    p_a_dep_fam_3:
        !Ponto antes de depositar
        pMov_Pega_Depos_Buffer := pPosição_Final_Buffer;
        pMov_Pega_Depos_Buffer.trans := pMov_Pega_Depos_Buffer.trans + pOfst_Z_Familia_3;
        IF (nPos_Buffer >= 13 AND nPos_Buffer <= 15) OR (nPos_Buffer >= 19 AND nPos_Buffer <= 21) OR (nPos_Buffer >= 25 AND nPos_Buffer <= 27) OR (nPos_Buffer >= 31 AND nPos_Buffer <=33) OR (nPos_Buffer >= 37 AND nPos_Buffer <= 39) OR (nPos_Buffer >= 43 AND nPos_Buffer <= 45) OR (nPos_Buffer >= 49 AND nPos_Buffer <= 51) OR (nPos_Buffer >= 55 AND nPos_Buffer <=57) OR (nPos_Buffer >= 61 AND nPos_Buffer <= 63) OR (nPos_Buffer >= 67 AND nPos_Buffer <= 69) OR (nPos_Buffer >= 73 AND nPos_Buffer <= 75) OR (nPos_Buffer >= 79 AND nPos_Buffer <= 81) OR (nPos_Buffer >= 85 AND nPos_Buffer <= 87) OR (nPos_Buffer >= 91 AND nPos_Buffer <= 93) OR (nPos_Buffer >= 97 AND nPos_Buffer <= 99) THEN
        MoveL pMov_Pega_Depos_Buffer, SMov_SuperFina, z10, tGarra \WObj:=wBuffer_Dir;
        GOTO p_ant_ag_3;
        ENDIF
        IF (nPos_Buffer >= 1 AND nPos_Buffer <= 9) THEN
        MoveL pMov_Pega_Depos_Buffer, SMov_SuperFina, z10, tGarra \WObj:=wBuffer_Front;
        GOTO p_ant_ag_3;
        ELSE
        MoveL pMov_Pega_Depos_Buffer, SMov_SuperFina, z10, tGarra \WObj:=wBuffer_Esq;
        ENDIF

    p_ant_ag_3:
        pMov_Pega_Depos_Buffer := pPosição_Final_Buffer;
        pMov_Pega_Depos_Buffer.trans := pMov_Pega_Depos_Buffer.trans + pOfst_Aprox_Final_Depos;
        IF (nPos_Buffer >= 13 AND nPos_Buffer <= 15) OR (nPos_Buffer >= 19 AND nPos_Buffer <= 21) OR (nPos_Buffer >= 25 AND nPos_Buffer <= 27) OR (nPos_Buffer >= 31 AND nPos_Buffer <=33) OR (nPos_Buffer >= 37 AND nPos_Buffer <= 39) OR (nPos_Buffer >= 43 AND nPos_Buffer <= 45) OR (nPos_Buffer >= 49 AND nPos_Buffer <= 51) OR (nPos_Buffer >= 55 AND nPos_Buffer <=57) OR (nPos_Buffer >= 61 AND nPos_Buffer <= 63) OR (nPos_Buffer >= 67 AND nPos_Buffer <= 69) OR (nPos_Buffer >= 73 AND nPos_Buffer <= 75) OR (nPos_Buffer >= 79 AND nPos_Buffer <= 81) OR (nPos_Buffer >= 85 AND nPos_Buffer <= 87) OR (nPos_Buffer >= 91 AND nPos_Buffer <= 93) OR (nPos_Buffer >= 97 AND nPos_Buffer <= 99) THEN
        MoveL pMov_Pega_Depos_Buffer, SMov_SuperFina, z1, tGarra \WObj:=wBuffer_Dir;
        GOTO p_depos_3;
        ENDIF
        IF (nPos_Buffer >= 1 AND nPos_Buffer <= 9) THEN
        MoveL pMov_Pega_Depos_Buffer, SMov_SuperFina, z1, tGarra \WObj:=wBuffer_Front;
        GOTO p_depos_3;
        ELSE
        MoveL pMov_Pega_Depos_Buffer, SMov_SuperFina, z1, tGarra \WObj:=wBuffer_Esq;
        ENDIF

    p_depos_3:
        !Destrava o produto
        GARRA_DestravarProduto;

        !Ponto final para depositar
        pMov_Pega_Depos_Buffer := pPosição_Final_Buffer;
        IF (nPos_Buffer >= 13 AND nPos_Buffer <= 15) OR (nPos_Buffer >= 19 AND nPos_Buffer <= 21) OR (nPos_Buffer >= 25 AND nPos_Buffer <= 27) OR (nPos_Buffer >= 31 AND nPos_Buffer <=33) OR (nPos_Buffer >= 37 AND nPos_Buffer <= 39) OR (nPos_Buffer >= 43 AND nPos_Buffer <= 45) OR (nPos_Buffer >= 49 AND nPos_Buffer <= 51) OR (nPos_Buffer >= 55 AND nPos_Buffer <=57) OR (nPos_Buffer >= 61 AND nPos_Buffer <= 63) OR (nPos_Buffer >= 67 AND nPos_Buffer <= 69) OR (nPos_Buffer >= 73 AND nPos_Buffer <= 75) OR (nPos_Buffer >= 79 AND nPos_Buffer <= 81) OR (nPos_Buffer >= 85 AND nPos_Buffer <= 87) OR (nPos_Buffer >= 91 AND nPos_Buffer <= 93) OR (nPos_Buffer >= 97 AND nPos_Buffer <= 99) THEN
        MoveL pMov_Pega_Depos_Buffer, SMov_SuperFina, fine, tGarra \WObj:=wBuffer_Dir;
        GOTO a_garra_3;
        ENDIF
        IF (nPos_Buffer >= 1 AND nPos_Buffer <= 9) THEN
        MoveL pMov_Pega_Depos_Buffer, SMov_SuperFina, fine, tGarra \WObj:=wBuffer_Front;
        GOTO a_garra_3;
        ELSE
        MoveL pMov_Pega_Depos_Buffer, SMov_SuperFina, fine, tGarra \WObj:=wBuffer_Esq;
        ENDIF


      a_garra_3:
        !Deposita Produto
        GARRA_AbrirGarra;

        GripLoad load0;

        !Movimento de Recuo
        AccSet nAcc_Mov_Geral, nRamp_Mov_Geral;
        pMov_Pega_Depos_Buffer := pPosição_Final_Buffer;
        pMov_Pega_Depos_Buffer.trans := pMov_Pega_Depos_Buffer.trans + pOfst_Acima_Berço_Buffer;
        IF (nPos_Buffer >= 13 AND nPos_Buffer <= 15) OR (nPos_Buffer >= 19 AND nPos_Buffer <= 21) OR (nPos_Buffer >= 25 AND nPos_Buffer <= 27) OR (nPos_Buffer >= 31 AND nPos_Buffer <=33) OR (nPos_Buffer >= 37 AND nPos_Buffer <= 39) OR (nPos_Buffer >= 43 AND nPos_Buffer <= 45) OR (nPos_Buffer >= 49 AND nPos_Buffer <= 51) OR (nPos_Buffer >= 55 AND nPos_Buffer <=57) OR (nPos_Buffer >= 61 AND nPos_Buffer <= 63) OR (nPos_Buffer >= 67 AND nPos_Buffer <= 69) OR (nPos_Buffer >= 73 AND nPos_Buffer <= 75) OR (nPos_Buffer >= 79 AND nPos_Buffer <= 81) OR (nPos_Buffer >= 85 AND nPos_Buffer <= 87) OR (nPos_Buffer >= 91 AND nPos_Buffer <= 93) OR (nPos_Buffer >= 97 AND nPos_Buffer <= 99) THEN
        MoveL pMov_Pega_Depos_Buffer, sMov_Aprox_Berço_Sem_Produto, z50, tGarra \WObj:=wBuffer_Dir;
        GOTO ad_buffer_3;
        ENDIF
        IF (nPos_Buffer >= 1 AND nPos_Buffer <= 9) THEN
        MoveL pMov_Pega_Depos_Buffer, sMov_Aprox_Berço_Sem_Produto, z50, tGarra \WObj:=wBuffer_Front;
        GOTO ad_buffer_3;
        ELSE
        MoveL pMov_Pega_Depos_Buffer, sMov_Aprox_Berço_Sem_Produto, z50, tGarra \WObj:=wBuffer_Esq;
        ENDIF

    ad_buffer_3:
        motionsup \On \TuneValue:= nSens_Colid_Mov_Geral;
        pMov_Pega_Depos_Buffer := pPosição_Final_Buffer;
        pMov_Pega_Depos_Buffer.trans := pMov_Pega_Depos_Buffer.trans + pOfst_Acima_Buffer_Sem_Produto;
        IF (nPos_Buffer >= 13 AND nPos_Buffer <= 15) OR (nPos_Buffer >= 19 AND nPos_Buffer <= 21) OR (nPos_Buffer >= 25 AND nPos_Buffer <= 27) OR (nPos_Buffer >= 31 AND nPos_Buffer <=33) OR (nPos_Buffer >= 37 AND nPos_Buffer <= 39) OR (nPos_Buffer >= 43 AND nPos_Buffer <= 45) OR (nPos_Buffer >= 49 AND nPos_Buffer <= 51) OR (nPos_Buffer >= 55 AND nPos_Buffer <=57) OR (nPos_Buffer >= 61 AND nPos_Buffer <= 63) OR (nPos_Buffer >= 67 AND nPos_Buffer <= 69) OR (nPos_Buffer >= 73 AND nPos_Buffer <= 75) OR (nPos_Buffer >= 79 AND nPos_Buffer <= 81) OR (nPos_Buffer >= 85 AND nPos_Buffer <= 87) OR (nPos_Buffer >= 91 AND nPos_Buffer <= 93) OR (nPos_Buffer >= 97 AND nPos_Buffer <= 99) THEN
        MoveL pMov_Pega_Depos_Buffer, sMov_Geral_Sem_Produto, z100, tGarra \WObj:=wBuffer_Dir;
        GOTO inposf_fam_3;
        ENDIF
        IF (nPos_Buffer >= 1 AND nPos_Buffer <= 9) THEN
        MoveL pMov_Pega_Depos_Buffer, sMov_Geral_Sem_Produto, z100, tGarra \WObj:=wBuffer_Front;
        GOTO inposf_fam_3;
        ELSE
        MoveL pMov_Pega_Depos_Buffer, sMov_Geral_Sem_Produto, z100, tGarra \WObj:=wBuffer_Esq;
        ENDIF
        GOTO inposf_fam_3;

inposf_fam_3:
        IF (nPos_Buffer >= 13 AND nPos_Buffer <= 15) OR (nPos_Buffer >= 19 AND nPos_Buffer <= 21) OR (nPos_Buffer >= 25 AND nPos_Buffer <= 27) OR (nPos_Buffer >= 31 AND nPos_Buffer <=33) OR (nPos_Buffer >= 37 AND nPos_Buffer <= 39) OR (nPos_Buffer >= 43 AND nPos_Buffer <= 45) OR (nPos_Buffer >= 49 AND nPos_Buffer <= 51) OR (nPos_Buffer >= 55 AND nPos_Buffer <=57) OR (nPos_Buffer >= 61 AND nPos_Buffer <= 63) OR (nPos_Buffer >= 67 AND nPos_Buffer <= 69) OR (nPos_Buffer >= 73 AND nPos_Buffer <= 75) OR (nPos_Buffer >= 79 AND nPos_Buffer <= 81) OR (nPos_Buffer >= 85 AND nPos_Buffer <= 87) OR (nPos_Buffer >= 91 AND nPos_Buffer <= 93) OR (nPos_Buffer >= 97 AND nPos_Buffer <= 99) THEN
        MoveAbsJ jposIntermedCentroMassa, sMov_Geral_Sem_Produto, z200, tGarra\WObj:=wBuffer_Dir;
        GOTO final;
        ENDIF
        IF (nPos_Buffer >= 1 AND nPos_Buffer <= 9) THEN
        MoveAbsJ jposIntermedCentroMassa, sMov_Geral_Sem_Produto, z200, tGarra\WObj:=wBuffer_Front;
        GOTO final;
        ELSE
        MoveAbsJ jposIntermedCentroMassa, sMov_Geral_Sem_Produto, z200, tGarra\WObj:=wBuffer_Esq;
        ENDIF
        GOTO final;

!*********************************************************************************************************************************************
!  PEGA PRODUTO NO BUFFER FAMILIA 3
!*********************************************************************************************************************************************

     pega_fam_3:
        !Ciclo para pegar peça no buffer

        GARRA_VerificarGarraVazia;
        !Abre Garra
        GARRA_DestravarProduto;
        GARRA_AbrirGarra;

        !Vai para posição intermediária no centro de massa
        AccSet nAcc_Mov_Geral, nRamp_Mov_Geral;

        IF (nPos_Buffer >= 13 AND nPos_Buffer <= 15) OR (nPos_Buffer >= 19 AND nPos_Buffer <= 21) OR (nPos_Buffer >= 25 AND nPos_Buffer <= 27) OR (nPos_Buffer >= 31 AND nPos_Buffer <=33) OR (nPos_Buffer >= 37 AND nPos_Buffer <= 39) OR (nPos_Buffer >= 43 AND nPos_Buffer <= 45) OR (nPos_Buffer >= 49 AND nPos_Buffer <= 51) OR (nPos_Buffer >= 55 AND nPos_Buffer <=57) OR (nPos_Buffer >= 61 AND nPos_Buffer <= 63) OR (nPos_Buffer >= 67 AND nPos_Buffer <= 69) OR (nPos_Buffer >= 73 AND nPos_Buffer <= 75) OR (nPos_Buffer >= 79 AND nPos_Buffer <= 81) OR (nPos_Buffer >= 85 AND nPos_Buffer <= 87) OR (nPos_Buffer >= 91 AND nPos_Buffer <= 93) OR (nPos_Buffer >= 97 AND nPos_Buffer <= 99) THEN
        pIntermedCentroMassa := pPosição_Final_Buffer;
	    jposIntermedCentroMassa := CalcJointT(pIntermedCentroMassa, tGarra \WObj:=wBuffer_Dir);
        jposIntermedCentroMassa.robax.rax_2 := jposRecolhidoEsteira.robax.rax_2;
        jposIntermedCentroMassa.robax.rax_3 := jposRecolhidoEsteira.robax.rax_3;
        jposIntermedCentroMassa.robax.rax_4 := jposRecolhidoEsteira.robax.rax_4;
        jposIntermedCentroMassa.robax.rax_5 := jposRecolhidoEsteira.robax.rax_5;

        MoveAbsJ jposIntermedCentroMassa, sMov_Geral_Sem_Produto, z200, tGarra\WObj:=wBuffer_Dir;
        GOTO inpegapos_fam_3;
        ENDIF

        IF (nPos_Buffer >= 1 AND nPos_Buffer <= 9) THEN
        pIntermedCentroMassa := pPosição_Final_Buffer;
	    jposIntermedCentroMassa := CalcJointT(pIntermedCentroMassa, tGarra \WObj:=wBuffer_Front);
        jposIntermedCentroMassa.robax.rax_2 := jposRecolhidoEsteira.robax.rax_2;
        jposIntermedCentroMassa.robax.rax_3 := jposRecolhidoEsteira.robax.rax_3;
        jposIntermedCentroMassa.robax.rax_4 := jposRecolhidoEsteira.robax.rax_4;
        jposIntermedCentroMassa.robax.rax_5 := jposRecolhidoEsteira.robax.rax_5;

        MoveAbsJ jposIntermedCentroMassa, sMov_Geral_Sem_Produto, z200, tGarra\WObj:=wBuffer_Front;
        GOTO inpegapos_fam_3;
        ELSE
        pIntermedCentroMassa := pPosição_Final_Buffer;
	    jposIntermedCentroMassa := CalcJointT(pIntermedCentroMassa, tGarra \WObj:=wBuffer_Esq);
        jposIntermedCentroMassa.robax.rax_2 := jposRecolhidoEsteira.robax.rax_2;
        jposIntermedCentroMassa.robax.rax_3 := jposRecolhidoEsteira.robax.rax_3;
        jposIntermedCentroMassa.robax.rax_4 := jposRecolhidoEsteira.robax.rax_4;
        jposIntermedCentroMassa.robax.rax_5 := jposRecolhidoEsteira.robax.rax_5;

        MoveAbsJ jposIntermedCentroMassa, sMov_Geral_Sem_Produto, z200, tGarra\WObj:=wBuffer_Esq;
        ENDIF

inpegapos_fam_3:
        !Ponto acima da posição
        pMov_Pega_Depos_Buffer := pPosição_Final_Buffer;
        pMov_Pega_Depos_Buffer.trans := pMov_Pega_Depos_Buffer.trans + pOfst_Acima_Buffer_Sem_Produto;
        IF (nPos_Buffer >= 13 AND nPos_Buffer <= 15) OR (nPos_Buffer >= 19 AND nPos_Buffer <= 21) OR (nPos_Buffer >= 25 AND nPos_Buffer <= 27) OR (nPos_Buffer >= 31 AND nPos_Buffer <=33) OR (nPos_Buffer >= 37 AND nPos_Buffer <= 39) OR (nPos_Buffer >= 43 AND nPos_Buffer <= 45) OR (nPos_Buffer >= 49 AND nPos_Buffer <= 51) OR (nPos_Buffer >= 55 AND nPos_Buffer <=57) OR (nPos_Buffer >= 61 AND nPos_Buffer <= 63) OR (nPos_Buffer >= 67 AND nPos_Buffer <= 69) OR (nPos_Buffer >= 73 AND nPos_Buffer <= 75) OR (nPos_Buffer >= 79 AND nPos_Buffer <= 81) OR (nPos_Buffer >= 85 AND nPos_Buffer <= 87) OR (nPos_Buffer >= 91 AND nPos_Buffer <= 93) OR (nPos_Buffer >= 97 AND nPos_Buffer <= 99) THEN
        MoveL pMov_Pega_Depos_Buffer, sMov_Geral_Sem_Produto, fine, tGarra \WObj:=wBuffer_Dir;
        GOTO  ap_berço_3;
        ENDIF
        IF (nPos_Buffer >= 1 AND nPos_Buffer <= 9) THEN
        MoveL pMov_Pega_Depos_Buffer, sMov_Geral_Sem_Produto, fine, tGarra \WObj:=wBuffer_Front;
        GOTO  ap_berço_3;
        ELSE
        MoveL pMov_Pega_Depos_Buffer, sMov_Geral_Sem_Produto, fine, tGarra \WObj:=wBuffer_Esq;
        ENDIF

      ap_berço_3:
        !Ponto acima do berço
        pMov_Pega_Depos_Buffer := pPosição_Final_Buffer;
        pMov_Pega_Depos_Buffer.trans := pMov_Pega_Depos_Buffer.trans + pOfst_Acima_Berço_Buffer;
        IF (nPos_Buffer >= 13 AND nPos_Buffer <= 15) OR (nPos_Buffer >= 19 AND nPos_Buffer <= 21) OR (nPos_Buffer >= 25 AND nPos_Buffer <= 27) OR (nPos_Buffer >= 31 AND nPos_Buffer <=33) OR (nPos_Buffer >= 37 AND nPos_Buffer <= 39) OR (nPos_Buffer >= 43 AND nPos_Buffer <= 45) OR (nPos_Buffer >= 49 AND nPos_Buffer <= 51) OR (nPos_Buffer >= 55 AND nPos_Buffer <=57) OR (nPos_Buffer >= 61 AND nPos_Buffer <= 63) OR (nPos_Buffer >= 67 AND nPos_Buffer <= 69) OR (nPos_Buffer >= 73 AND nPos_Buffer <= 75) OR (nPos_Buffer >= 79 AND nPos_Buffer <= 81) OR (nPos_Buffer >= 85 AND nPos_Buffer <= 87) OR (nPos_Buffer >= 91 AND nPos_Buffer <= 93) OR (nPos_Buffer >= 97 AND nPos_Buffer <= 99) THEN
        MoveL pMov_Pega_Depos_Buffer, sMov_Aprox_Berço_Sem_Produto, z100, tGarra \WObj:=wBuffer_Dir;
        GOTO  pp_aprox_3;
        ENDIF
        IF (nPos_Buffer >= 1 AND nPos_Buffer <= 9) THEN
        MoveL pMov_Pega_Depos_Buffer, sMov_Aprox_Berço_Sem_Produto, z100, tGarra \WObj:=wBuffer_Front;
        GOTO  pp_aprox_3;
        ELSE
        MoveL pMov_Pega_Depos_Buffer, sMov_Aprox_Berço_Sem_Produto, z100, tGarra \WObj:=wBuffer_Esq;
        ENDIF

    pp_aprox_3:
        !Ponto de aproximação
        motionsup \On \TuneValue:= nSens_Colid_Aprox;
        pMov_Pega_Depos_Buffer := pPosição_Final_Buffer;
        pMov_Pega_Depos_Buffer.trans := pMov_Pega_Depos_Buffer.trans + pOfst_Aprox_Pega_Depos_Buffer;
        IF (nPos_Buffer >= 13 AND nPos_Buffer <= 15) OR (nPos_Buffer >= 19 AND nPos_Buffer <= 21) OR (nPos_Buffer >= 25 AND nPos_Buffer <= 27) OR (nPos_Buffer >= 31 AND nPos_Buffer <=33) OR (nPos_Buffer >= 37 AND nPos_Buffer <= 39) OR (nPos_Buffer >= 43 AND nPos_Buffer <= 45) OR (nPos_Buffer >= 49 AND nPos_Buffer <= 51) OR (nPos_Buffer >= 55 AND nPos_Buffer <=57) OR (nPos_Buffer >= 61 AND nPos_Buffer <= 63) OR (nPos_Buffer >= 67 AND nPos_Buffer <= 69) OR (nPos_Buffer >= 73 AND nPos_Buffer <= 75) OR (nPos_Buffer >= 79 AND nPos_Buffer <= 81) OR (nPos_Buffer >= 85 AND nPos_Buffer <= 87) OR (nPos_Buffer >= 91 AND nPos_Buffer <= 93) OR (nPos_Buffer >= 97 AND nPos_Buffer <= 99) THEN
        MoveL pMov_Pega_Depos_Buffer, SMov_Fina, z50, tGarra \WObj:=wBuffer_Dir;
        GOTO  p_peça_3;
        ENDIF
        IF (nPos_Buffer >= 1 AND nPos_Buffer <= 9) THEN
        MoveL pMov_Pega_Depos_Buffer, SMov_Fina, z50, tGarra \WObj:=wBuffer_Front;
        GOTO  p_peça_3;
        ELSE
        MoveL pMov_Pega_Depos_Buffer, SMov_Fina, z50, tGarra \WObj:=wBuffer_Esq;
        ENDIF

    p_peça_3:
        !Ponto de pega
        pMov_Pega_Depos_Buffer := pPosição_Final_Buffer;
        IF (nPos_Buffer >= 13 AND nPos_Buffer <= 15) OR (nPos_Buffer >= 19 AND nPos_Buffer <= 21) OR (nPos_Buffer >= 25 AND nPos_Buffer <= 27) OR (nPos_Buffer >= 31 AND nPos_Buffer <=33) OR (nPos_Buffer >= 37 AND nPos_Buffer <= 39) OR (nPos_Buffer >= 43 AND nPos_Buffer <= 45) OR (nPos_Buffer >= 49 AND nPos_Buffer <= 51) OR (nPos_Buffer >= 55 AND nPos_Buffer <=57) OR (nPos_Buffer >= 61 AND nPos_Buffer <= 63) OR (nPos_Buffer >= 67 AND nPos_Buffer <= 69) OR (nPos_Buffer >= 73 AND nPos_Buffer <= 75) OR (nPos_Buffer >= 79 AND nPos_Buffer <= 81) OR (nPos_Buffer >= 85 AND nPos_Buffer <= 87) OR (nPos_Buffer >= 91 AND nPos_Buffer <= 93) OR (nPos_Buffer >= 97 AND nPos_Buffer <= 99) THEN
        MoveL pMov_Pega_Depos_Buffer, SMov_SuperFina, fine, tGarra \WObj:=wBuffer_Dir;
        GOTO f_garra_3;
        ENDIF
        IF (nPos_Buffer >= 1 AND nPos_Buffer <= 9) THEN
        MoveL pMov_Pega_Depos_Buffer, SMov_SuperFina, fine, tGarra \WObj:=wBuffer_Front;
        GOTO f_garra_3;
        ELSE
        MoveL pMov_Pega_Depos_Buffer, SMov_SuperFina, fine, tGarra \WObj:=wBuffer_Esq;
        ENDIF

    f_garra_3:
        !Pega Produto
        GARRA_FecharGarra;

        GripLoad lFamilia_3;

        AccSet nAcc_Mov_Pega_Depos, nRamp_Mov_Pega_Depos;
        pMov_Pega_Depos_Buffer := pPosição_Final_Buffer;
        pMov_Pega_Depos_Buffer.trans := pMov_Pega_Depos_Buffer.trans + pOfst_Aprox_Inicial_Pega;
        IF (nPos_Buffer >= 13 AND nPos_Buffer <= 15) OR (nPos_Buffer >= 19 AND nPos_Buffer <= 21) OR (nPos_Buffer >= 25 AND nPos_Buffer <= 27) OR (nPos_Buffer >= 31 AND nPos_Buffer <=33) OR (nPos_Buffer >= 37 AND nPos_Buffer <= 39) OR (nPos_Buffer >= 43 AND nPos_Buffer <= 45) OR (nPos_Buffer >= 49 AND nPos_Buffer <= 51) OR (nPos_Buffer >= 55 AND nPos_Buffer <=57) OR (nPos_Buffer >= 61 AND nPos_Buffer <= 63) OR (nPos_Buffer >= 67 AND nPos_Buffer <= 69) OR (nPos_Buffer >= 73 AND nPos_Buffer <= 75) OR (nPos_Buffer >= 79 AND nPos_Buffer <= 81) OR (nPos_Buffer >= 85 AND nPos_Buffer <= 87) OR (nPos_Buffer >= 91 AND nPos_Buffer <= 93) OR (nPos_Buffer >= 97 AND nPos_Buffer <= 99) THEN
        MoveL pMov_Pega_Depos_Buffer, SMov_SuperFina, z1, tGarra \WObj:=wBuffer_Dir;
        GOTO   tp_ac_3;
        ENDIF
        IF (nPos_Buffer >= 1 AND nPos_Buffer <= 9) THEN
        MoveL pMov_Pega_Depos_Buffer, SMov_SuperFina, z1, tGarra \WObj:=wBuffer_Front;
        GOTO   tp_ac_3;
        ELSE
        MoveL pMov_Pega_Depos_Buffer, SMov_SuperFina, z1, tGarra \WObj:=wBuffer_Esq;
        ENDIF

    tp_ac_3:
        !Trava o produto
        GARRA_TravarProduto;

        !Movimento 1 de Recuo
        pMov_Pega_Depos_Buffer := pPosição_Final_Buffer;
        pMov_Pega_Depos_Buffer.trans := pMov_Pega_Depos_Buffer.trans + pOfst_Z_Familia_3;
        IF (nPos_Buffer >= 13 AND nPos_Buffer <= 15) OR (nPos_Buffer >= 19 AND nPos_Buffer <= 21) OR (nPos_Buffer >= 25 AND nPos_Buffer <= 27) OR (nPos_Buffer >= 31 AND nPos_Buffer <=33) OR (nPos_Buffer >= 37 AND nPos_Buffer <= 39) OR (nPos_Buffer >= 43 AND nPos_Buffer <= 45) OR (nPos_Buffer >= 49 AND nPos_Buffer <= 51) OR (nPos_Buffer >= 55 AND nPos_Buffer <=57) OR (nPos_Buffer >= 61 AND nPos_Buffer <= 63) OR (nPos_Buffer >= 67 AND nPos_Buffer <= 69) OR (nPos_Buffer >= 73 AND nPos_Buffer <= 75) OR (nPos_Buffer >= 79 AND nPos_Buffer <= 81) OR (nPos_Buffer >= 85 AND nPos_Buffer <= 87) OR (nPos_Buffer >= 91 AND nPos_Buffer <= 93) OR (nPos_Buffer >= 97 AND nPos_Buffer <= 99) THEN
        MoveL pMov_Pega_Depos_Buffer, SMov_SuperFina, z10, tGarra \WObj:=wBuffer_Dir;
        GOTO   m_1_p_fam_3;
        ENDIF
        IF (nPos_Buffer >= 1 AND nPos_Buffer <= 9) THEN
        MoveL pMov_Pega_Depos_Buffer, SMov_SuperFina, z10, tGarra \WObj:=wBuffer_Front;
        GOTO   m_1_p_fam_3;
        ELSE
        MoveL pMov_Pega_Depos_Buffer, SMov_SuperFina, z10, tGarra \WObj:=wBuffer_Esq;
        ENDIF

    m_1_p_fam_3:
        !Movimento 2 de Recuo
        pMov_Pega_Depos_Buffer := pPosição_Final_Buffer;
        pMov_Pega_Depos_Buffer.trans := pMov_Pega_Depos_Buffer.trans + pOfst_ZY_Familia_3;
        IF (nPos_Buffer >= 13 AND nPos_Buffer <= 15) OR (nPos_Buffer >= 19 AND nPos_Buffer <= 21) OR (nPos_Buffer >= 25 AND nPos_Buffer <= 27) OR (nPos_Buffer >= 31 AND nPos_Buffer <=33) OR (nPos_Buffer >= 37 AND nPos_Buffer <= 39) OR (nPos_Buffer >= 43 AND nPos_Buffer <= 45) OR (nPos_Buffer >= 49 AND nPos_Buffer <= 51) OR (nPos_Buffer >= 55 AND nPos_Buffer <=57) OR (nPos_Buffer >= 61 AND nPos_Buffer <= 63) OR (nPos_Buffer >= 67 AND nPos_Buffer <= 69) OR (nPos_Buffer >= 73 AND nPos_Buffer <= 75) OR (nPos_Buffer >= 79 AND nPos_Buffer <= 81) OR (nPos_Buffer >= 85 AND nPos_Buffer <= 87) OR (nPos_Buffer >= 91 AND nPos_Buffer <= 93) OR (nPos_Buffer >= 97 AND nPos_Buffer <= 99) THEN
        MoveL pMov_Pega_Depos_Buffer, SMov_SuperFina, z10, tGarra \WObj:=wBuffer_Dir;
        GOTO   m_2_p_fam_3;
        ENDIF
        IF (nPos_Buffer >= 1 AND nPos_Buffer <= 9) THEN
        MoveL pMov_Pega_Depos_Buffer, SMov_SuperFina, z10, tGarra \WObj:=wBuffer_Front;
        GOTO   m_2_p_fam_3;
        ELSE
        MoveL pMov_Pega_Depos_Buffer, SMov_SuperFina, z10, tGarra \WObj:=wBuffer_Esq;
        ENDIF

    m_2_p_fam_3:
        !Movimento de Recuo
        pMov_Pega_Depos_Buffer := pPosição_Final_Buffer;
        pMov_Pega_Depos_Buffer.trans := pMov_Pega_Depos_Buffer.trans + pOfst_Acima_Berço_Buffer;
        IF (nPos_Buffer >= 13 AND nPos_Buffer <= 15) OR (nPos_Buffer >= 19 AND nPos_Buffer <= 21) OR (nPos_Buffer >= 25 AND nPos_Buffer <= 27) OR (nPos_Buffer >= 31 AND nPos_Buffer <=33) OR (nPos_Buffer >= 37 AND nPos_Buffer <= 39) OR (nPos_Buffer >= 43 AND nPos_Buffer <= 45) OR (nPos_Buffer >= 49 AND nPos_Buffer <= 51) OR (nPos_Buffer >= 55 AND nPos_Buffer <=57) OR (nPos_Buffer >= 61 AND nPos_Buffer <= 63) OR (nPos_Buffer >= 67 AND nPos_Buffer <= 69) OR (nPos_Buffer >= 73 AND nPos_Buffer <= 75) OR (nPos_Buffer >= 79 AND nPos_Buffer <= 81) OR (nPos_Buffer >= 85 AND nPos_Buffer <= 87) OR (nPos_Buffer >= 91 AND nPos_Buffer <= 93) OR (nPos_Buffer >= 97 AND nPos_Buffer <= 99) THEN
        MoveL pMov_Pega_Depos_Buffer, SMov_Levanta_Com_Produto, z100, tGarra \WObj:=wBuffer_Dir;
        GOTO  ap_buffer_3;
        ENDIF
        IF (nPos_Buffer >= 1 AND nPos_Buffer <= 9) THEN
        MoveL pMov_Pega_Depos_Buffer, SMov_Levanta_Com_Produto, z100, tGarra \WObj:=wBuffer_Front;
        GOTO  ap_buffer_3;
        ELSE
        MoveL pMov_Pega_Depos_Buffer, SMov_Levanta_Com_Produto, z100, tGarra \WObj:=wBuffer_Esq;
        ENDIF

    ap_buffer_3:
        AccSet nAcc_Mov_Geral, nRamp_Mov_Geral;
        motionsup \On \TuneValue:= nSens_Colid_Mov_Geral;
        pMov_Pega_Depos_Buffer := pPosição_Final_Buffer;
        pMov_Pega_Depos_Buffer.trans := pMov_Pega_Depos_Buffer.trans + pOfst_Acima_Buffer;
        IF (nPos_Buffer >= 13 AND nPos_Buffer <= 15) OR (nPos_Buffer >= 19 AND nPos_Buffer <= 21) OR (nPos_Buffer >= 25 AND nPos_Buffer <= 27) OR (nPos_Buffer >= 31 AND nPos_Buffer <=33) OR (nPos_Buffer >= 37 AND nPos_Buffer <= 39) OR (nPos_Buffer >= 43 AND nPos_Buffer <= 45) OR (nPos_Buffer >= 49 AND nPos_Buffer <= 51) OR (nPos_Buffer >= 55 AND nPos_Buffer <=57) OR (nPos_Buffer >= 61 AND nPos_Buffer <= 63) OR (nPos_Buffer >= 67 AND nPos_Buffer <= 69) OR (nPos_Buffer >= 73 AND nPos_Buffer <= 75) OR (nPos_Buffer >= 79 AND nPos_Buffer <= 81) OR (nPos_Buffer >= 85 AND nPos_Buffer <= 87) OR (nPos_Buffer >= 91 AND nPos_Buffer <= 93) OR (nPos_Buffer >= 97 AND nPos_Buffer <= 99) THEN
        MoveL pMov_Pega_Depos_Buffer, sMov_Geral_Com_Produto, z100, tGarra \WObj:=wBuffer_Dir;
        GOTO  inpegaposf_fam_3;
        ENDIF
        IF (nPos_Buffer >= 1 AND nPos_Buffer <= 9) THEN
        MoveL pMov_Pega_Depos_Buffer, sMov_Geral_Com_Produto, z100, tGarra \WObj:=wBuffer_Front;
        GOTO  inpegaposf_fam_3;
        ELSE
        MoveL pMov_Pega_Depos_Buffer, sMov_Geral_Com_Produto, z100, tGarra \WObj:=wBuffer_Esq;
        ENDIF
        GOTO inpegaposf_fam_3;

    inpegaposf_fam_3:
        IF (nPos_Buffer >= 13 AND nPos_Buffer <= 15) OR (nPos_Buffer >= 19 AND nPos_Buffer <= 21) OR (nPos_Buffer >= 25 AND nPos_Buffer <= 27) OR (nPos_Buffer >= 31 AND nPos_Buffer <=33) OR (nPos_Buffer >= 37 AND nPos_Buffer <= 39) OR (nPos_Buffer >= 43 AND nPos_Buffer <= 45) OR (nPos_Buffer >= 49 AND nPos_Buffer <= 51) OR (nPos_Buffer >= 55 AND nPos_Buffer <=57) OR (nPos_Buffer >= 61 AND nPos_Buffer <= 63) OR (nPos_Buffer >= 67 AND nPos_Buffer <= 69) OR (nPos_Buffer >= 73 AND nPos_Buffer <= 75) OR (nPos_Buffer >= 79 AND nPos_Buffer <= 81) OR (nPos_Buffer >= 85 AND nPos_Buffer <= 87) OR (nPos_Buffer >= 91 AND nPos_Buffer <= 93) OR (nPos_Buffer >= 97 AND nPos_Buffer <= 99) THEN
        MoveAbsJ jposIntermedCentroMassa, sMov_Geral_Com_Produto, z200, tGarra\WObj:=wBuffer_Dir;
        GOTO  final;
        ENDIF
        IF (nPos_Buffer >= 1 AND nPos_Buffer <= 9) THEN
        MoveAbsJ jposIntermedCentroMassa, sMov_Geral_Com_Produto, z200, tGarra\WObj:=wBuffer_Front;
        GOTO  final;
        ELSE
        MoveAbsJ jposIntermedCentroMassa, sMov_Geral_Com_Produto, z200, tGarra\WObj:=wBuffer_Esq;
        ENDIF
        GOTO final;

!*********************************************************************************************************************************************
!  DEPOSITA PRODUTO NO BUFFER FAMILIA 4
!*********************************************************************************************************************************************

    deposita_fam_4:
        !Ciclo para depositar peça no buffer

        !Ponto intermediario centro de massa
        AccSet nAcc_Mov_Geral, nRamp_Mov_Geral;
        IF (nPos_Buffer >= 13 AND nPos_Buffer <= 15) OR (nPos_Buffer >= 19 AND nPos_Buffer <= 21) OR (nPos_Buffer >= 25 AND nPos_Buffer <= 27) OR (nPos_Buffer >= 31 AND nPos_Buffer <=33) OR (nPos_Buffer >= 37 AND nPos_Buffer <= 39) OR (nPos_Buffer >= 43 AND nPos_Buffer <= 45) OR (nPos_Buffer >= 49 AND nPos_Buffer <= 51) OR (nPos_Buffer >= 55 AND nPos_Buffer <=57) OR (nPos_Buffer >= 61 AND nPos_Buffer <= 63) OR (nPos_Buffer >= 67 AND nPos_Buffer <= 69) OR (nPos_Buffer >= 73 AND nPos_Buffer <= 75) OR (nPos_Buffer >= 79 AND nPos_Buffer <= 81) OR (nPos_Buffer >= 85 AND nPos_Buffer <= 87) OR (nPos_Buffer >= 91 AND nPos_Buffer <= 93) OR (nPos_Buffer >= 97 AND nPos_Buffer <= 99) THEN
        pIntermedCentroMassa := pPosição_Final_Buffer;
	    jposIntermedCentroMassa := CalcJointT(pIntermedCentroMassa, tGarra \WObj:=wBuffer_Dir);
        jposIntermedCentroMassa.robax.rax_2 := jposRecolhidoEsteira.robax.rax_2;
        jposIntermedCentroMassa.robax.rax_3 := jposRecolhidoEsteira.robax.rax_3;
        jposIntermedCentroMassa.robax.rax_4 := jposRecolhidoEsteira.robax.rax_4;
        jposIntermedCentroMassa.robax.rax_5 := jposRecolhidoEsteira.robax.rax_5;

        MoveAbsJ jposIntermedCentroMassa, sMov_Geral_Com_Produto, z200, tGarra\WObj:=wBuffer_Dir;
        GOTO inpos_fam_4;
        ENDIF

        IF (nPos_Buffer >= 1 AND nPos_Buffer <= 9) THEN
        pIntermedCentroMassa := pPosição_Final_Buffer;
	    jposIntermedCentroMassa := CalcJointT(pIntermedCentroMassa, tGarra \WObj:=wBuffer_Front);
        jposIntermedCentroMassa.robax.rax_2 := jposRecolhidoEsteira.robax.rax_2;
        jposIntermedCentroMassa.robax.rax_3 := jposRecolhidoEsteira.robax.rax_3;
        jposIntermedCentroMassa.robax.rax_4 := jposRecolhidoEsteira.robax.rax_4;
        jposIntermedCentroMassa.robax.rax_5 := jposRecolhidoEsteira.robax.rax_5;

        MoveAbsJ jposIntermedCentroMassa, sMov_Geral_Com_Produto, z200, tGarra\WObj:=wBuffer_Front;
        GOTO inpos_fam_4;
        ELSE
        pIntermedCentroMassa := pPosição_Final_Buffer;
	    jposIntermedCentroMassa := CalcJointT(pIntermedCentroMassa, tGarra \WObj:=wBuffer_Esq);
        jposIntermedCentroMassa.robax.rax_2 := jposRecolhidoEsteira.robax.rax_2;
        jposIntermedCentroMassa.robax.rax_3 := jposRecolhidoEsteira.robax.rax_3;
        jposIntermedCentroMassa.robax.rax_4 := jposRecolhidoEsteira.robax.rax_4;
        jposIntermedCentroMassa.robax.rax_5 := jposRecolhidoEsteira.robax.rax_5;

        MoveAbsJ jposIntermedCentroMassa, sMov_Geral_Com_Produto, z200, tGarra\WObj:=wBuffer_Esq;
        ENDIF

inpos_fam_4:
        !Ponto acima da posição
        pMov_Pega_Depos_Buffer := pPosição_Final_Buffer;
        pMov_Pega_Depos_Buffer.trans := pMov_Pega_Depos_Buffer.trans + pOfst_Acima_Buffer;
        IF (nPos_Buffer >= 13 AND nPos_Buffer <= 15) OR (nPos_Buffer >= 19 AND nPos_Buffer <= 21) OR (nPos_Buffer >= 25 AND nPos_Buffer <= 27) OR (nPos_Buffer >= 31 AND nPos_Buffer <=33) OR (nPos_Buffer >= 37 AND nPos_Buffer <= 39) OR (nPos_Buffer >= 43 AND nPos_Buffer <= 45) OR (nPos_Buffer >= 49 AND nPos_Buffer <= 51) OR (nPos_Buffer >= 55 AND nPos_Buffer <=57) OR (nPos_Buffer >= 61 AND nPos_Buffer <= 63) OR (nPos_Buffer >= 67 AND nPos_Buffer <= 69) OR (nPos_Buffer >= 73 AND nPos_Buffer <= 75) OR (nPos_Buffer >= 79 AND nPos_Buffer <= 81) OR (nPos_Buffer >= 85 AND nPos_Buffer <= 87) OR (nPos_Buffer >= 91 AND nPos_Buffer <= 93) OR (nPos_Buffer >= 97 AND nPos_Buffer <= 99) THEN
        MoveJ pMov_Pega_Depos_Buffer, sMov_Geral_Com_Produto, fine, tGarra \WObj:=wBuffer_Dir;
        GOTO verifica_fam_4;
        ENDIF
        IF (nPos_Buffer >= 1 AND nPos_Buffer <= 9) THEN
        MoveJ pMov_Pega_Depos_Buffer, sMov_Geral_Com_Produto, fine, tGarra \WObj:=wBuffer_Front;
        GOTO verifica_fam_4;
        ELSE
        MoveJ pMov_Pega_Depos_Buffer, sMov_Geral_Com_Produto, fine, tGarra \WObj:=wBuffer_Esq;
        ENDIF

    verifica_fam_4:
        !Verifica se já existe peça na posição selecionada
        IF DInput (DI_Pres_Peça_Berço_1) = 0 AND DInput (DI_Pres_Peça_Berço_2) = 1 GOTO a_berço_4;

        !Caso exista produto no berço selecionado
        TPWrite "Já existe um produto na posição "\num:= nPos_Buffer;
        SetDO PN_OUT_Produto_Existente, 1;
        Stop;
        GOTO inpos_fam_4;

    a_berço_4:
        SetDO PN_OUT_Produto_Existente, 0;

        !Ponto acima do berço
        pMov_Pega_Depos_Buffer := pPosição_Final_Buffer;
        pMov_Pega_Depos_Buffer.trans := pMov_Pega_Depos_Buffer.trans + pOfst_Acima_Berço_Buffer + pOfst_ZY_Familia_4;
        IF (nPos_Buffer >= 13 AND nPos_Buffer <= 15) OR (nPos_Buffer >= 19 AND nPos_Buffer <= 21) OR (nPos_Buffer >= 25 AND nPos_Buffer <= 27) OR (nPos_Buffer >= 31 AND nPos_Buffer <=33) OR (nPos_Buffer >= 37 AND nPos_Buffer <= 39) OR (nPos_Buffer >= 43 AND nPos_Buffer <= 45) OR (nPos_Buffer >= 49 AND nPos_Buffer <= 51) OR (nPos_Buffer >= 55 AND nPos_Buffer <=57) OR (nPos_Buffer >= 61 AND nPos_Buffer <= 63) OR (nPos_Buffer >= 67 AND nPos_Buffer <= 69) OR (nPos_Buffer >= 73 AND nPos_Buffer <= 75) OR (nPos_Buffer >= 79 AND nPos_Buffer <= 81) OR (nPos_Buffer >= 85 AND nPos_Buffer <= 87) OR (nPos_Buffer >= 91 AND nPos_Buffer <= 93) OR (nPos_Buffer >= 97 AND nPos_Buffer <= 99) THEN
        MoveL pMov_Pega_Depos_Buffer, sMov_Aprox_Berço_Com_Produto, z50, tGarra \WObj:=wBuffer_Dir;
        GOTO p_aprox_4;
        ENDIF
        IF (nPos_Buffer >= 1 AND nPos_Buffer <= 9) THEN
        MoveL pMov_Pega_Depos_Buffer, sMov_Aprox_Berço_Com_Produto, z50, tGarra \WObj:=wBuffer_Front;
        GOTO p_aprox_4;
        ELSE
        MoveL pMov_Pega_Depos_Buffer, sMov_Aprox_Berço_Com_Produto, z50, tGarra \WObj:=wBuffer_Esq;
        ENDIF

    p_aprox_4:
        !Ponto de aproximação
        AccSet nAcc_Mov_Pega_Depos, nRamp_Mov_Pega_Depos;
        motionsup \On \TuneValue:= nSens_Colid_Aprox;
        pMov_Pega_Depos_Buffer := pPosição_Final_Buffer;
        pMov_Pega_Depos_Buffer.trans := pMov_Pega_Depos_Buffer.trans + pOfst_ZY_Familia_4;
        IF (nPos_Buffer >= 13 AND nPos_Buffer <= 15) OR (nPos_Buffer >= 19 AND nPos_Buffer <= 21) OR (nPos_Buffer >= 25 AND nPos_Buffer <= 27) OR (nPos_Buffer >= 31 AND nPos_Buffer <=33) OR (nPos_Buffer >= 37 AND nPos_Buffer <= 39) OR (nPos_Buffer >= 43 AND nPos_Buffer <= 45) OR (nPos_Buffer >= 49 AND nPos_Buffer <= 51) OR (nPos_Buffer >= 55 AND nPos_Buffer <=57) OR (nPos_Buffer >= 61 AND nPos_Buffer <= 63) OR (nPos_Buffer >= 67 AND nPos_Buffer <= 69) OR (nPos_Buffer >= 73 AND nPos_Buffer <= 75) OR (nPos_Buffer >= 79 AND nPos_Buffer <= 81) OR (nPos_Buffer >= 85 AND nPos_Buffer <= 87) OR (nPos_Buffer >= 91 AND nPos_Buffer <= 93) OR (nPos_Buffer >= 97 AND nPos_Buffer <= 99) THEN
        MoveL pMov_Pega_Depos_Buffer, SMov_Fina, z10, tGarra \WObj:=wBuffer_Dir;
        GOTO p_a_dep_fam_4;
        ENDIF
        IF (nPos_Buffer >= 1 AND nPos_Buffer <= 9) THEN
        MoveL pMov_Pega_Depos_Buffer, SMov_Fina, z10, tGarra \WObj:=wBuffer_Front;
        GOTO p_a_dep_fam_4;
        ELSE
        MoveL pMov_Pega_Depos_Buffer, SMov_Fina, z10, tGarra \WObj:=wBuffer_Esq;
        ENDIF

    p_a_dep_fam_4:
        !Ponto antes de depositar
        pMov_Pega_Depos_Buffer := pPosição_Final_Buffer;
        pMov_Pega_Depos_Buffer.trans := pMov_Pega_Depos_Buffer.trans + pOfst_Z_Familia_4;
        IF (nPos_Buffer >= 13 AND nPos_Buffer <= 15) OR (nPos_Buffer >= 19 AND nPos_Buffer <= 21) OR (nPos_Buffer >= 25 AND nPos_Buffer <= 27) OR (nPos_Buffer >= 31 AND nPos_Buffer <=33) OR (nPos_Buffer >= 37 AND nPos_Buffer <= 39) OR (nPos_Buffer >= 43 AND nPos_Buffer <= 45) OR (nPos_Buffer >= 49 AND nPos_Buffer <= 51) OR (nPos_Buffer >= 55 AND nPos_Buffer <=57) OR (nPos_Buffer >= 61 AND nPos_Buffer <= 63) OR (nPos_Buffer >= 67 AND nPos_Buffer <= 69) OR (nPos_Buffer >= 73 AND nPos_Buffer <= 75) OR (nPos_Buffer >= 79 AND nPos_Buffer <= 81) OR (nPos_Buffer >= 85 AND nPos_Buffer <= 87) OR (nPos_Buffer >= 91 AND nPos_Buffer <= 93) OR (nPos_Buffer >= 97 AND nPos_Buffer <= 99) THEN
        MoveL pMov_Pega_Depos_Buffer, SMov_SuperFina, z10, tGarra \WObj:=wBuffer_Dir;
        GOTO p_ant_ag_4;
        ENDIF
        IF (nPos_Buffer >= 1 AND nPos_Buffer <= 9) THEN
        MoveL pMov_Pega_Depos_Buffer, SMov_SuperFina, z10, tGarra \WObj:=wBuffer_Front;
        GOTO p_ant_ag_4;
        ELSE
        MoveL pMov_Pega_Depos_Buffer, SMov_SuperFina, z10, tGarra \WObj:=wBuffer_Esq;
        ENDIF

    p_ant_ag_4:
        pMov_Pega_Depos_Buffer := pPosição_Final_Buffer;
        pMov_Pega_Depos_Buffer.trans := pMov_Pega_Depos_Buffer.trans + pOfst_Aprox_Final_Depos;
        IF (nPos_Buffer >= 13 AND nPos_Buffer <= 15) OR (nPos_Buffer >= 19 AND nPos_Buffer <= 21) OR (nPos_Buffer >= 25 AND nPos_Buffer <= 27) OR (nPos_Buffer >= 31 AND nPos_Buffer <=33) OR (nPos_Buffer >= 37 AND nPos_Buffer <= 39) OR (nPos_Buffer >= 43 AND nPos_Buffer <= 45) OR (nPos_Buffer >= 49 AND nPos_Buffer <= 51) OR (nPos_Buffer >= 55 AND nPos_Buffer <=57) OR (nPos_Buffer >= 61 AND nPos_Buffer <= 63) OR (nPos_Buffer >= 67 AND nPos_Buffer <= 69) OR (nPos_Buffer >= 73 AND nPos_Buffer <= 75) OR (nPos_Buffer >= 79 AND nPos_Buffer <= 81) OR (nPos_Buffer >= 85 AND nPos_Buffer <= 87) OR (nPos_Buffer >= 91 AND nPos_Buffer <= 93) OR (nPos_Buffer >= 97 AND nPos_Buffer <= 99) THEN
        MoveL pMov_Pega_Depos_Buffer, SMov_SuperFina, z1, tGarra \WObj:=wBuffer_Dir;
        GOTO p_depos_4;
        ENDIF
       IF (nPos_Buffer >= 1 AND nPos_Buffer <= 9) THEN
        MoveL pMov_Pega_Depos_Buffer, SMov_SuperFina, z1, tGarra \WObj:=wBuffer_Front;
        GOTO p_depos_4;
        ELSE
        MoveL pMov_Pega_Depos_Buffer, SMov_SuperFina, z1, tGarra \WObj:=wBuffer_Esq;
        ENDIF

    p_depos_4:
        !Destrava o produto
        GARRA_DestravarProduto;

        !Ponto final para depositar
        pMov_Pega_Depos_Buffer := pPosição_Final_Buffer;
        IF (nPos_Buffer >= 13 AND nPos_Buffer <= 15) OR (nPos_Buffer >= 19 AND nPos_Buffer <= 21) OR (nPos_Buffer >= 25 AND nPos_Buffer <= 27) OR (nPos_Buffer >= 31 AND nPos_Buffer <=33) OR (nPos_Buffer >= 37 AND nPos_Buffer <= 39) OR (nPos_Buffer >= 43 AND nPos_Buffer <= 45) OR (nPos_Buffer >= 49 AND nPos_Buffer <= 51) OR (nPos_Buffer >= 55 AND nPos_Buffer <=57) OR (nPos_Buffer >= 61 AND nPos_Buffer <= 63) OR (nPos_Buffer >= 67 AND nPos_Buffer <= 69) OR (nPos_Buffer >= 73 AND nPos_Buffer <= 75) OR (nPos_Buffer >= 79 AND nPos_Buffer <= 81) OR (nPos_Buffer >= 85 AND nPos_Buffer <= 87) OR (nPos_Buffer >= 91 AND nPos_Buffer <= 93) OR (nPos_Buffer >= 97 AND nPos_Buffer <= 99) THEN
        MoveL pMov_Pega_Depos_Buffer, SMov_SuperFina, fine, tGarra \WObj:=wBuffer_Dir;
        GOTO a_garra_4;
        ENDIF
        IF (nPos_Buffer >= 1 AND nPos_Buffer <= 9) THEN
        MoveL pMov_Pega_Depos_Buffer, SMov_SuperFina, fine, tGarra \WObj:=wBuffer_Front;
        GOTO a_garra_4;
        ELSE
        MoveL pMov_Pega_Depos_Buffer, SMov_SuperFina, fine, tGarra \WObj:=wBuffer_Esq;
        ENDIF


      a_garra_4:
        !Deposita Produto
        GARRA_AbrirGarra;

        GripLoad load0;

        !Movimento de Recuo
        pMov_Pega_Depos_Buffer := pPosição_Final_Buffer;
        pMov_Pega_Depos_Buffer.trans := pMov_Pega_Depos_Buffer.trans + pOfst_Acima_Berço_Buffer;
        IF (nPos_Buffer >= 13 AND nPos_Buffer <= 15) OR (nPos_Buffer >= 19 AND nPos_Buffer <= 21) OR (nPos_Buffer >= 25 AND nPos_Buffer <= 27) OR (nPos_Buffer >= 31 AND nPos_Buffer <=33) OR (nPos_Buffer >= 37 AND nPos_Buffer <= 39) OR (nPos_Buffer >= 43 AND nPos_Buffer <= 45) OR (nPos_Buffer >= 49 AND nPos_Buffer <= 51) OR (nPos_Buffer >= 55 AND nPos_Buffer <=57) OR (nPos_Buffer >= 61 AND nPos_Buffer <= 63) OR (nPos_Buffer >= 67 AND nPos_Buffer <= 69) OR (nPos_Buffer >= 73 AND nPos_Buffer <= 75) OR (nPos_Buffer >= 79 AND nPos_Buffer <= 81) OR (nPos_Buffer >= 85 AND nPos_Buffer <= 87) OR (nPos_Buffer >= 91 AND nPos_Buffer <= 93) OR (nPos_Buffer >= 97 AND nPos_Buffer <= 99) THEN
        MoveL pMov_Pega_Depos_Buffer, sMov_Aprox_Berço_Sem_Produto, z50, tGarra \WObj:=wBuffer_Dir;
        GOTO ad_buffer_4;
        ENDIF
        IF (nPos_Buffer >= 1 AND nPos_Buffer <= 9) THEN
        MoveJ pMov_Pega_Depos_Buffer, sMov_Geral_Sem_Produto, z50, tGarra \WObj:=wBuffer_Front;
        GOTO ad_buffer_4;
        ELSE
        MoveJ pMov_Pega_Depos_Buffer, sMov_Aprox_Berço_Sem_Produto, z50, tGarra \WObj:=wBuffer_Esq;
        ENDIF

    ad_buffer_4:
        AccSet nAcc_Mov_Geral, nRamp_Mov_Geral;
        motionsup \On \TuneValue:= nSens_Colid_Mov_Geral;
        pMov_Pega_Depos_Buffer := pPosição_Final_Buffer;
        pMov_Pega_Depos_Buffer.trans := pMov_Pega_Depos_Buffer.trans + pOfst_Acima_Buffer_Sem_Produto;
        IF (nPos_Buffer >= 13 AND nPos_Buffer <= 15) OR (nPos_Buffer >= 19 AND nPos_Buffer <= 21) OR (nPos_Buffer >= 25 AND nPos_Buffer <= 27) OR (nPos_Buffer >= 31 AND nPos_Buffer <=33) OR (nPos_Buffer >= 37 AND nPos_Buffer <= 39) OR (nPos_Buffer >= 43 AND nPos_Buffer <= 45) OR (nPos_Buffer >= 49 AND nPos_Buffer <= 51) OR (nPos_Buffer >= 55 AND nPos_Buffer <=57) OR (nPos_Buffer >= 61 AND nPos_Buffer <= 63) OR (nPos_Buffer >= 67 AND nPos_Buffer <= 69) OR (nPos_Buffer >= 73 AND nPos_Buffer <= 75) OR (nPos_Buffer >= 79 AND nPos_Buffer <= 81) OR (nPos_Buffer >= 85 AND nPos_Buffer <= 87) OR (nPos_Buffer >= 91 AND nPos_Buffer <= 93) OR (nPos_Buffer >= 97 AND nPos_Buffer <= 99) THEN
        MoveL pMov_Pega_Depos_Buffer, sMov_Geral_Sem_Produto, z50, tGarra \WObj:=wBuffer_Dir;
        GOTO inposf_fam_4;
        ENDIF
        IF (nPos_Buffer >= 1 AND nPos_Buffer <= 9) THEN
        MoveL pMov_Pega_Depos_Buffer, sMov_Geral_Sem_Produto, z50, tGarra \WObj:=wBuffer_Front;
        GOTO inposf_fam_4;
        ELSE
        MoveL pMov_Pega_Depos_Buffer, sMov_Geral_Sem_Produto, z50, tGarra \WObj:=wBuffer_Esq;
        ENDIF
        GOTO inposf_fam_4;

    inposf_fam_4:
        IF (nPos_Buffer >= 13 AND nPos_Buffer <= 15) OR (nPos_Buffer >= 19 AND nPos_Buffer <= 21) OR (nPos_Buffer >= 25 AND nPos_Buffer <= 27) OR (nPos_Buffer >= 31 AND nPos_Buffer <=33) OR (nPos_Buffer >= 37 AND nPos_Buffer <= 39) OR (nPos_Buffer >= 43 AND nPos_Buffer <= 45) OR (nPos_Buffer >= 49 AND nPos_Buffer <= 51) OR (nPos_Buffer >= 55 AND nPos_Buffer <=57) OR (nPos_Buffer >= 61 AND nPos_Buffer <= 63) OR (nPos_Buffer >= 67 AND nPos_Buffer <= 69) OR (nPos_Buffer >= 73 AND nPos_Buffer <= 75) OR (nPos_Buffer >= 79 AND nPos_Buffer <= 81) OR (nPos_Buffer >= 85 AND nPos_Buffer <= 87) OR (nPos_Buffer >= 91 AND nPos_Buffer <= 93) OR (nPos_Buffer >= 97 AND nPos_Buffer <= 99) THEN
        MoveAbsJ jposIntermedCentroMassa, sMov_Geral_Sem_Produto, z200, tGarra\WObj:=wBuffer_Dir;
        GOTO final;
        ENDIF
        IF (nPos_Buffer >= 1 AND nPos_Buffer <= 9) THEN
        MoveAbsJ jposIntermedCentroMassa, sMov_Geral_Sem_Produto, z200, tGarra\WObj:=wBuffer_Front;
        GOTO final;
        ELSE
        MoveAbsJ jposIntermedCentroMassa, sMov_Geral_Sem_Produto, z200, tGarra\WObj:=wBuffer_Esq;
        ENDIF
        GOTO final;

!*********************************************************************************************************************************************
!  PEGA PRODUTO NO BUFFER FAMILIA 4
!*********************************************************************************************************************************************

     pega_fam_4:
        !Ciclo para pegar peça no buffer

        GARRA_VerificarGarraVazia;
        !Abre Garra
        GARRA_DestravarProduto;
        GARRA_AbrirGarra;

        !Ponto acima da posição
        AccSet nAcc_Mov_Geral, nRamp_Mov_Geral;

        IF (nPos_Buffer >= 13 AND nPos_Buffer <= 15) OR (nPos_Buffer >= 19 AND nPos_Buffer <= 21) OR (nPos_Buffer >= 25 AND nPos_Buffer <= 27) OR (nPos_Buffer >= 31 AND nPos_Buffer <=33) OR (nPos_Buffer >= 37 AND nPos_Buffer <= 39) OR (nPos_Buffer >= 43 AND nPos_Buffer <= 45) OR (nPos_Buffer >= 49 AND nPos_Buffer <= 51) OR (nPos_Buffer >= 55 AND nPos_Buffer <=57) OR (nPos_Buffer >= 61 AND nPos_Buffer <= 63) OR (nPos_Buffer >= 67 AND nPos_Buffer <= 69) OR (nPos_Buffer >= 73 AND nPos_Buffer <= 75) OR (nPos_Buffer >= 79 AND nPos_Buffer <= 81) OR (nPos_Buffer >= 85 AND nPos_Buffer <= 87) OR (nPos_Buffer >= 91 AND nPos_Buffer <= 93) OR (nPos_Buffer >= 97 AND nPos_Buffer <= 99) THEN
        pIntermedCentroMassa := pPosição_Final_Buffer;
	    jposIntermedCentroMassa := CalcJointT(pIntermedCentroMassa, tGarra \WObj:=wBuffer_Dir);
        jposIntermedCentroMassa.robax.rax_2 := jposRecolhidoEsteira.robax.rax_2;
        jposIntermedCentroMassa.robax.rax_3 := jposRecolhidoEsteira.robax.rax_3;
        jposIntermedCentroMassa.robax.rax_4 := jposRecolhidoEsteira.robax.rax_4;
        jposIntermedCentroMassa.robax.rax_5 := jposRecolhidoEsteira.robax.rax_5;

        MoveAbsJ jposIntermedCentroMassa, sMov_Geral_Sem_Produto, z200, tGarra\WObj:=wBuffer_Dir;
        GOTO inpegapos_fam_4;
        ENDIF

        IF (nPos_Buffer >= 1 AND nPos_Buffer <= 9) THEN
        pIntermedCentroMassa := pPosição_Final_Buffer;
	    jposIntermedCentroMassa := CalcJointT(pIntermedCentroMassa, tGarra \WObj:=wBuffer_Front);
        jposIntermedCentroMassa.robax.rax_2 := jposRecolhidoEsteira.robax.rax_2;
        jposIntermedCentroMassa.robax.rax_3 := jposRecolhidoEsteira.robax.rax_3;
        jposIntermedCentroMassa.robax.rax_4 := jposRecolhidoEsteira.robax.rax_4;
        jposIntermedCentroMassa.robax.rax_5 := jposRecolhidoEsteira.robax.rax_5;

        MoveAbsJ jposIntermedCentroMassa, sMov_Geral_Sem_Produto, z200, tGarra\WObj:=wBuffer_Front;
        GOTO inpegapos_fam_4;
        ELSE
        pIntermedCentroMassa := pPosição_Final_Buffer;
	    jposIntermedCentroMassa := CalcJointT(pIntermedCentroMassa, tGarra \WObj:=wBuffer_Esq);
        jposIntermedCentroMassa.robax.rax_2 := jposRecolhidoEsteira.robax.rax_2;
        jposIntermedCentroMassa.robax.rax_3 := jposRecolhidoEsteira.robax.rax_3;
        jposIntermedCentroMassa.robax.rax_4 := jposRecolhidoEsteira.robax.rax_4;
        jposIntermedCentroMassa.robax.rax_5 := jposRecolhidoEsteira.robax.rax_5;

        MoveAbsJ jposIntermedCentroMassa, sMov_Geral_Sem_Produto, z200, tGarra\WObj:=wBuffer_Esq;
        ENDIF

    inpegapos_fam_4:
        pMov_Pega_Depos_Buffer := pPosição_Final_Buffer;
        pMov_Pega_Depos_Buffer.trans := pMov_Pega_Depos_Buffer.trans + pOfst_Acima_Buffer;
        IF (nPos_Buffer >= 13 AND nPos_Buffer <= 15) OR (nPos_Buffer >= 19 AND nPos_Buffer <= 21) OR (nPos_Buffer >= 25 AND nPos_Buffer <= 27) OR (nPos_Buffer >= 31 AND nPos_Buffer <=33) OR (nPos_Buffer >= 37 AND nPos_Buffer <= 39) OR (nPos_Buffer >= 43 AND nPos_Buffer <= 45) OR (nPos_Buffer >= 49 AND nPos_Buffer <= 51) OR (nPos_Buffer >= 55 AND nPos_Buffer <=57) OR (nPos_Buffer >= 61 AND nPos_Buffer <= 63) OR (nPos_Buffer >= 67 AND nPos_Buffer <= 69) OR (nPos_Buffer >= 73 AND nPos_Buffer <= 75) OR (nPos_Buffer >= 79 AND nPos_Buffer <= 81) OR (nPos_Buffer >= 85 AND nPos_Buffer <= 87) OR (nPos_Buffer >= 91 AND nPos_Buffer <= 93) OR (nPos_Buffer >= 97 AND nPos_Buffer <= 99) THEN
        MoveL pMov_Pega_Depos_Buffer, sMov_Geral_Sem_Produto, fine, tGarra \WObj:=wBuffer_Dir;
        GOTO  ap_berço_4;
        ENDIF
        IF (nPos_Buffer >= 1 AND nPos_Buffer <= 9) THEN
        MoveL pMov_Pega_Depos_Buffer, sMov_Geral_Sem_Produto, fine, tGarra \WObj:=wBuffer_Front;
        GOTO  ap_berço_4;
        ELSE
        MoveL pMov_Pega_Depos_Buffer, sMov_Geral_Sem_Produto, fine, tGarra \WObj:=wBuffer_Esq;
        ENDIF

    ap_berço_4:
        !Ponto acima do berço
        pMov_Pega_Depos_Buffer := pPosição_Final_Buffer;
        pMov_Pega_Depos_Buffer.trans := pMov_Pega_Depos_Buffer.trans + pOfst_Acima_Berço_Buffer;
        IF (nPos_Buffer >= 13 AND nPos_Buffer <= 15) OR (nPos_Buffer >= 19 AND nPos_Buffer <= 21) OR (nPos_Buffer >= 25 AND nPos_Buffer <= 27) OR (nPos_Buffer >= 31 AND nPos_Buffer <=33) OR (nPos_Buffer >= 37 AND nPos_Buffer <= 39) OR (nPos_Buffer >= 43 AND nPos_Buffer <= 45) OR (nPos_Buffer >= 49 AND nPos_Buffer <= 51) OR (nPos_Buffer >= 55 AND nPos_Buffer <=57) OR (nPos_Buffer >= 61 AND nPos_Buffer <= 63) OR (nPos_Buffer >= 67 AND nPos_Buffer <= 69) OR (nPos_Buffer >= 73 AND nPos_Buffer <= 75) OR (nPos_Buffer >= 79 AND nPos_Buffer <= 81) OR (nPos_Buffer >= 85 AND nPos_Buffer <= 87) OR (nPos_Buffer >= 91 AND nPos_Buffer <= 93) OR (nPos_Buffer >= 97 AND nPos_Buffer <= 99) THEN
        MoveL pMov_Pega_Depos_Buffer, sMov_Aprox_Berço_Sem_Produto, z50, tGarra \WObj:=wBuffer_Dir;
        GOTO  pp_aprox_4;
        ENDIF
        IF (nPos_Buffer >= 1 AND nPos_Buffer <= 9) THEN
        MoveL pMov_Pega_Depos_Buffer, sMov_Aprox_Berço_Sem_Produto, z50, tGarra \WObj:=wBuffer_Front;
        GOTO  pp_aprox_4;
        ELSE
        MoveL pMov_Pega_Depos_Buffer, sMov_Aprox_Berço_Sem_Produto, z50, tGarra \WObj:=wBuffer_Esq;
        ENDIF

    pp_aprox_4:
        !Ponto de aproximação
        motionsup \On \TuneValue:= nSens_Colid_Aprox;
        pMov_Pega_Depos_Buffer := pPosição_Final_Buffer;
        pMov_Pega_Depos_Buffer.trans := pMov_Pega_Depos_Buffer.trans + pOfst_Aprox_Pega_Depos_Buffer;
        IF (nPos_Buffer >= 13 AND nPos_Buffer <= 15) OR (nPos_Buffer >= 19 AND nPos_Buffer <= 21) OR (nPos_Buffer >= 25 AND nPos_Buffer <= 27) OR (nPos_Buffer >= 31 AND nPos_Buffer <=33) OR (nPos_Buffer >= 37 AND nPos_Buffer <= 39) OR (nPos_Buffer >= 43 AND nPos_Buffer <= 45) OR (nPos_Buffer >= 49 AND nPos_Buffer <= 51) OR (nPos_Buffer >= 55 AND nPos_Buffer <=57) OR (nPos_Buffer >= 61 AND nPos_Buffer <= 63) OR (nPos_Buffer >= 67 AND nPos_Buffer <= 69) OR (nPos_Buffer >= 73 AND nPos_Buffer <= 75) OR (nPos_Buffer >= 79 AND nPos_Buffer <= 81) OR (nPos_Buffer >= 85 AND nPos_Buffer <= 87) OR (nPos_Buffer >= 91 AND nPos_Buffer <= 93) OR (nPos_Buffer >= 97 AND nPos_Buffer <= 99) THEN
        MoveL pMov_Pega_Depos_Buffer, SMov_Fina, z50, tGarra \WObj:=wBuffer_Dir;
        GOTO  p_peça_4;
        ENDIF
        IF (nPos_Buffer >= 1 AND nPos_Buffer <= 9) THEN
        MoveL pMov_Pega_Depos_Buffer, SMov_Fina, z50, tGarra \WObj:=wBuffer_Front;
        GOTO  p_peça_4;
        ELSE
        MoveL pMov_Pega_Depos_Buffer, SMov_Fina, z50, tGarra \WObj:=wBuffer_Esq;
        ENDIF

    p_peça_4:
        !Ponto de pega
        pMov_Pega_Depos_Buffer := pPosição_Final_Buffer;
        IF (nPos_Buffer >= 13 AND nPos_Buffer <= 15) OR (nPos_Buffer >= 19 AND nPos_Buffer <= 21) OR (nPos_Buffer >= 25 AND nPos_Buffer <= 27) OR (nPos_Buffer >= 31 AND nPos_Buffer <=33) OR (nPos_Buffer >= 37 AND nPos_Buffer <= 39) OR (nPos_Buffer >= 43 AND nPos_Buffer <= 45) OR (nPos_Buffer >= 49 AND nPos_Buffer <= 51) OR (nPos_Buffer >= 55 AND nPos_Buffer <=57) OR (nPos_Buffer >= 61 AND nPos_Buffer <= 63) OR (nPos_Buffer >= 67 AND nPos_Buffer <= 69) OR (nPos_Buffer >= 73 AND nPos_Buffer <= 75) OR (nPos_Buffer >= 79 AND nPos_Buffer <= 81) OR (nPos_Buffer >= 85 AND nPos_Buffer <= 87) OR (nPos_Buffer >= 91 AND nPos_Buffer <= 93) OR (nPos_Buffer >= 97 AND nPos_Buffer <= 99) THEN
        MoveL pMov_Pega_Depos_Buffer, SMov_SuperFina, fine, tGarra \WObj:=wBuffer_Dir;
        GOTO f_garra_4;
        ENDIF
        IF (nPos_Buffer >= 1 AND nPos_Buffer <= 9) THEN
        MoveJ pMov_Pega_Depos_Buffer, SMov_SuperFina, fine, tGarra \WObj:=wBuffer_Front;
        GOTO f_garra_4;
        ELSE
        MoveJ pMov_Pega_Depos_Buffer, SMov_SuperFina, fine, tGarra \WObj:=wBuffer_Esq;
        ENDIF

    f_garra_4:
        !Pega Produto
        GARRA_FecharGarra;

        GripLoad lFamilia_4;

        AccSet nAcc_Mov_Pega_Depos, nRamp_Mov_Pega_Depos;
        pMov_Pega_Depos_Buffer := pPosição_Final_Buffer;
        pMov_Pega_Depos_Buffer.trans := pMov_Pega_Depos_Buffer.trans + pOfst_Aprox_Inicial_Pega;
        IF (nPos_Buffer >= 13 AND nPos_Buffer <= 15) OR (nPos_Buffer >= 19 AND nPos_Buffer <= 21) OR (nPos_Buffer >= 25 AND nPos_Buffer <= 27) OR (nPos_Buffer >= 31 AND nPos_Buffer <=33) OR (nPos_Buffer >= 37 AND nPos_Buffer <= 39) OR (nPos_Buffer >= 43 AND nPos_Buffer <= 45) OR (nPos_Buffer >= 49 AND nPos_Buffer <= 51) OR (nPos_Buffer >= 55 AND nPos_Buffer <=57) OR (nPos_Buffer >= 61 AND nPos_Buffer <= 63) OR (nPos_Buffer >= 67 AND nPos_Buffer <= 69) OR (nPos_Buffer >= 73 AND nPos_Buffer <= 75) OR (nPos_Buffer >= 79 AND nPos_Buffer <= 81) OR (nPos_Buffer >= 85 AND nPos_Buffer <= 87) OR (nPos_Buffer >= 91 AND nPos_Buffer <= 93) OR (nPos_Buffer >= 97 AND nPos_Buffer <= 99) THEN
        MoveL pMov_Pega_Depos_Buffer, SMov_SuperFina, z1, tGarra \WObj:=wBuffer_Dir;
        GOTO   tp_ac_4;
        ENDIF
        IF (nPos_Buffer >= 1 AND nPos_Buffer <= 9) THEN
        MoveJ pMov_Pega_Depos_Buffer, SMov_SuperFina, z1, tGarra \WObj:=wBuffer_Front;
        GOTO   tp_ac_4;
        ELSE
        MoveJ pMov_Pega_Depos_Buffer, SMov_SuperFina, z1, tGarra \WObj:=wBuffer_Esq;
        ENDIF

    tp_ac_4:
        !Trava o produto
        GARRA_TravarProduto;

        !Movimento 1 de Recuo
        pMov_Pega_Depos_Buffer := pPosição_Final_Buffer;
        pMov_Pega_Depos_Buffer.trans := pMov_Pega_Depos_Buffer.trans + pOfst_Z_Familia_4;
        IF (nPos_Buffer >= 13 AND nPos_Buffer <= 15) OR (nPos_Buffer >= 19 AND nPos_Buffer <= 21) OR (nPos_Buffer >= 25 AND nPos_Buffer <= 27) OR (nPos_Buffer >= 31 AND nPos_Buffer <=33) OR (nPos_Buffer >= 37 AND nPos_Buffer <= 39) OR (nPos_Buffer >= 43 AND nPos_Buffer <= 45) OR (nPos_Buffer >= 49 AND nPos_Buffer <= 51) OR (nPos_Buffer >= 55 AND nPos_Buffer <=57) OR (nPos_Buffer >= 61 AND nPos_Buffer <= 63) OR (nPos_Buffer >= 67 AND nPos_Buffer <= 69) OR (nPos_Buffer >= 73 AND nPos_Buffer <= 75) OR (nPos_Buffer >= 79 AND nPos_Buffer <= 81) OR (nPos_Buffer >= 85 AND nPos_Buffer <= 87) OR (nPos_Buffer >= 91 AND nPos_Buffer <= 93) OR (nPos_Buffer >= 97 AND nPos_Buffer <= 99) THEN
        MoveL pMov_Pega_Depos_Buffer, SMov_SuperFina, z10, tGarra \WObj:=wBuffer_Dir;
        GOTO   m_1_p_fam_4;
        ENDIF
        IF (nPos_Buffer >= 1 AND nPos_Buffer <= 9) THEN
        MoveJ pMov_Pega_Depos_Buffer, SMov_SuperFina, z10, tGarra \WObj:=wBuffer_Front;
        GOTO   m_1_p_fam_4;
        ELSE
        MoveJ pMov_Pega_Depos_Buffer, SMov_SuperFina, z10, tGarra \WObj:=wBuffer_Esq;
        ENDIF

    m_1_p_fam_4:
        !Movimento 2 de Recuo
        pMov_Pega_Depos_Buffer := pPosição_Final_Buffer;
        pMov_Pega_Depos_Buffer.trans := pMov_Pega_Depos_Buffer.trans + pOfst_ZY_Familia_4;
        IF (nPos_Buffer >= 13 AND nPos_Buffer <= 15) OR (nPos_Buffer >= 19 AND nPos_Buffer <= 21) OR (nPos_Buffer >= 25 AND nPos_Buffer <= 27) OR (nPos_Buffer >= 31 AND nPos_Buffer <=33) OR (nPos_Buffer >= 37 AND nPos_Buffer <= 39) OR (nPos_Buffer >= 43 AND nPos_Buffer <= 45) OR (nPos_Buffer >= 49 AND nPos_Buffer <= 51) OR (nPos_Buffer >= 55 AND nPos_Buffer <=57) OR (nPos_Buffer >= 61 AND nPos_Buffer <= 63) OR (nPos_Buffer >= 67 AND nPos_Buffer <= 69) OR (nPos_Buffer >= 73 AND nPos_Buffer <= 75) OR (nPos_Buffer >= 79 AND nPos_Buffer <= 81) OR (nPos_Buffer >= 85 AND nPos_Buffer <= 87) OR (nPos_Buffer >= 91 AND nPos_Buffer <= 93) OR (nPos_Buffer >= 97 AND nPos_Buffer <= 99) THEN
        MoveL pMov_Pega_Depos_Buffer, SMov_SuperFina, z10, tGarra \WObj:=wBuffer_Dir;
        GOTO   m_2_p_fam_4;
        ENDIF
        IF (nPos_Buffer >= 1 AND nPos_Buffer <= 9) THEN
        MoveJ pMov_Pega_Depos_Buffer, SMov_SuperFina, z10, tGarra \WObj:=wBuffer_Front;
        GOTO   m_2_p_fam_4;
        ELSE
        MoveJ pMov_Pega_Depos_Buffer, SMov_SuperFina, z10, tGarra \WObj:=wBuffer_Esq;
        ENDIF

    m_2_p_fam_4:
        !Movimento de Recuo
        pMov_Pega_Depos_Buffer := pPosição_Final_Buffer;
        pMov_Pega_Depos_Buffer.trans := pMov_Pega_Depos_Buffer.trans + pOfst_Acima_Berço_Buffer;
        IF (nPos_Buffer >= 13 AND nPos_Buffer <= 15) OR (nPos_Buffer >= 19 AND nPos_Buffer <= 21) OR (nPos_Buffer >= 25 AND nPos_Buffer <= 27) OR (nPos_Buffer >= 31 AND nPos_Buffer <=33) OR (nPos_Buffer >= 37 AND nPos_Buffer <= 39) OR (nPos_Buffer >= 43 AND nPos_Buffer <= 45) OR (nPos_Buffer >= 49 AND nPos_Buffer <= 51) OR (nPos_Buffer >= 55 AND nPos_Buffer <=57) OR (nPos_Buffer >= 61 AND nPos_Buffer <= 63) OR (nPos_Buffer >= 67 AND nPos_Buffer <= 69) OR (nPos_Buffer >= 73 AND nPos_Buffer <= 75) OR (nPos_Buffer >= 79 AND nPos_Buffer <= 81) OR (nPos_Buffer >= 85 AND nPos_Buffer <= 87) OR (nPos_Buffer >= 91 AND nPos_Buffer <= 93) OR (nPos_Buffer >= 97 AND nPos_Buffer <= 99) THEN
        MoveL pMov_Pega_Depos_Buffer, SMov_Levanta_Com_Produto, z50, tGarra \WObj:=wBuffer_Dir;
        GOTO  ap_buffer_4;
        ENDIF
        IF (nPos_Buffer >= 1 AND nPos_Buffer <= 9) THEN
        MoveJ pMov_Pega_Depos_Buffer, SMov_Levanta_Com_Produto, z50, tGarra \WObj:=wBuffer_Front;
        GOTO  ap_buffer_4;
        ELSE
        MoveJ pMov_Pega_Depos_Buffer, SMov_Levanta_Com_Produto, z50, tGarra \WObj:=wBuffer_Esq;
        ENDIF

    ap_buffer_4:
        AccSet nAcc_Mov_Geral, nRamp_Mov_Geral;
        motionsup \On \TuneValue:= nSens_Colid_Mov_Geral;
        pMov_Pega_Depos_Buffer := pPosição_Final_Buffer;
        pMov_Pega_Depos_Buffer.trans := pMov_Pega_Depos_Buffer.trans + pOfst_Acima_Buffer;
        IF (nPos_Buffer >= 13 AND nPos_Buffer <= 15) OR (nPos_Buffer >= 19 AND nPos_Buffer <= 21) OR (nPos_Buffer >= 25 AND nPos_Buffer <= 27) OR (nPos_Buffer >= 31 AND nPos_Buffer <=33) OR (nPos_Buffer >= 37 AND nPos_Buffer <= 39) OR (nPos_Buffer >= 43 AND nPos_Buffer <= 45) OR (nPos_Buffer >= 49 AND nPos_Buffer <= 51) OR (nPos_Buffer >= 55 AND nPos_Buffer <=57) OR (nPos_Buffer >= 61 AND nPos_Buffer <= 63) OR (nPos_Buffer >= 67 AND nPos_Buffer <= 69) OR (nPos_Buffer >= 73 AND nPos_Buffer <= 75) OR (nPos_Buffer >= 79 AND nPos_Buffer <= 81) OR (nPos_Buffer >= 85 AND nPos_Buffer <= 87) OR (nPos_Buffer >= 91 AND nPos_Buffer <= 93) OR (nPos_Buffer >= 97 AND nPos_Buffer <= 99) THEN
        MoveL pMov_Pega_Depos_Buffer, sMov_Geral_Com_Produto, z50, tGarra \WObj:=wBuffer_Dir;
        GOTO  inpegaposf_fam_4;
        ENDIF
        IF (nPos_Buffer >= 1 AND nPos_Buffer <= 9) THEN
        MoveJ pMov_Pega_Depos_Buffer, sMov_Geral_Com_Produto, z50, tGarra \WObj:=wBuffer_Front;
        GOTO  inpegaposf_fam_4;
        ELSE
        MoveJ pMov_Pega_Depos_Buffer, sMov_Geral_Com_Produto, z50, tGarra \WObj:=wBuffer_Esq;
        ENDIF
        GOTO inpegaposf_fam_4;

    inpegaposf_fam_4:
        IF (nPos_Buffer >= 13 AND nPos_Buffer <= 15) OR (nPos_Buffer >= 19 AND nPos_Buffer <= 21) OR (nPos_Buffer >= 25 AND nPos_Buffer <= 27) OR (nPos_Buffer >= 31 AND nPos_Buffer <=33) OR (nPos_Buffer >= 37 AND nPos_Buffer <= 39) OR (nPos_Buffer >= 43 AND nPos_Buffer <= 45) OR (nPos_Buffer >= 49 AND nPos_Buffer <= 51) OR (nPos_Buffer >= 55 AND nPos_Buffer <=57) OR (nPos_Buffer >= 61 AND nPos_Buffer <= 63) OR (nPos_Buffer >= 67 AND nPos_Buffer <= 69) OR (nPos_Buffer >= 73 AND nPos_Buffer <= 75) OR (nPos_Buffer >= 79 AND nPos_Buffer <= 81) OR (nPos_Buffer >= 85 AND nPos_Buffer <= 87) OR (nPos_Buffer >= 91 AND nPos_Buffer <= 93) OR (nPos_Buffer >= 97 AND nPos_Buffer <= 99) THEN
        MoveAbsJ jposIntermedCentroMassa, sMov_Geral_Com_Produto, z200, tGarra\WObj:=wBuffer_Dir;
        GOTO  final;
        ENDIF
        IF (nPos_Buffer >= 1 AND nPos_Buffer <= 9) THEN
        MoveAbsJ jposIntermedCentroMassa, sMov_Geral_Com_Produto, z200, tGarra\WObj:=wBuffer_Front;
        GOTO  final;
        ELSE
        MoveAbsJ jposIntermedCentroMassa, sMov_Geral_Com_Produto, z200, tGarra\WObj:=wBuffer_Esq;
        ENDIF
        GOTO final;

    final:
        IF GInput (PN_IN_Numero_Programa) = 3 THEN
        !Vai Posição de Trabalho
        MoveJ pPosição_Trabalho, sMov_Geral_Sem_Produto, z200, tGarra \WObj:=wobj0;
        GOTO fim;
        ENDIF

        IF (GInput (PN_IN_Numero_Programa) = 4 AND (nPos_Buffer >= 13 AND nPos_Buffer <= 15) OR (nPos_Buffer >= 19 AND nPos_Buffer <= 21) OR (nPos_Buffer >= 25 AND nPos_Buffer <= 27) OR (nPos_Buffer >= 31 AND nPos_Buffer <=33) OR (nPos_Buffer >= 37 AND nPos_Buffer <= 39) OR (nPos_Buffer >= 43 AND nPos_Buffer <= 45) OR (nPos_Buffer >= 49 AND nPos_Buffer <= 51) OR (nPos_Buffer >= 55 AND nPos_Buffer <=57) OR (nPos_Buffer >= 61 AND nPos_Buffer <= 63) OR (nPos_Buffer >= 67 AND nPos_Buffer <= 69) OR (nPos_Buffer >= 73 AND nPos_Buffer <= 75) OR (nPos_Buffer >= 79 AND nPos_Buffer <= 81) OR (nPos_Buffer >= 85 AND nPos_Buffer <= 87) OR (nPos_Buffer >= 91 AND nPos_Buffer <= 93) OR (nPos_Buffer >= 97 AND nPos_Buffer <= 99)) GOTO fim;

        !Vai Posição de Trabalho
        MoveJ pPosição_Trabalho, sMov_Geral_Com_Produto, z200, tGarra \WObj:=wobj0;

    fim:
        !Avisa clp que finalizou rotina
        ComunicaCLP;

	ENDPROC

    !*************************************************************************************************************************
    !Troca de Dados CLP
    !*************************************************************************************************************************
    PROC ComunicaCLP()
        !Avisa clp que finalizou rotina
        Set PN_OUT_Programa_Finalizado;
        WaitGI PN_IN_Numero_Programa, 0;
        Reset PN_OUT_Programa_Finalizado;
    ENDPROC

    !*************************************************************************************************************************
    !Reset de flags
    !*************************************************************************************************************************
    PROC ResetFlags()
        SetDO \Sync, PN_OUT_Solicita_Abertura, 0;
        SetDO \Sync, PN_OUT_Solicita_Fecha_Garra, 0;
        SetDO\Sync, PN_OUT_Programa_Finalizado, 0;
    ENDPROC

    !*************************************************************************************************************************
    !Retorna wObjData (Frame) de um index qualquer do Buffer
    !*************************************************************************************************************************
     FUNC wobjdata GetWObjBuffer(Num i)

         !Area C (Robô de Costas para Esteira, à Direita
            IF (i >= 13 AND i <= 15) OR (i >= 19 AND i <= 21) OR (i >= 25 AND i <= 27) OR (i >= 31 AND i <=33) OR (i >= 37 AND i <= 39) OR (i >= 43 AND i <= 45) OR (i >= 49 AND i <= 51) OR (i >= 55 AND i <=57) OR (i >= 61 AND i <= 63) OR (i >= 67 AND i <= 69) OR (i >= 73 AND i <= 75) OR (i >= 79 AND i <= 81) OR (i >= 85 AND i <= 87) OR (i >= 91 AND i <= 93) OR (i >= 97 AND i <= 99) THEN
                Return wBuffer_Dir;

            !Area B (Robô de Costas para Esteira, à sua Frente
            ELSEIF (i >= 1 AND i <= 9) THEN
                RETURN wBuffer_Front;

            !Area A (Robô de Costas para Esteira, à sua Esquerda
            ELSE
                RETURN wBuffer_Esq;
            ENDIF
     ENDFUNC

    !*************************************************************************************************************************
    !Retorna área de um index qualquer do Buffer
    !*************************************************************************************************************************
     FUNC string GetAreaBuffer(Num i)

         !Area C (Robô de Costas para Esteira, à Direita
            IF (i >= 13 AND i <= 15) OR (i >= 19 AND i <= 21) OR (i >= 25 AND i <= 27) OR (i >= 31 AND i <=33) OR (i >= 37 AND i <= 39) OR (i >= 43 AND i <= 45) OR (i >= 49 AND i <= 51) OR (i >= 55 AND i <=57) OR (i >= 61 AND i <= 63) OR (i >= 67 AND i <= 69) OR (i >= 73 AND i <= 75) OR (i >= 79 AND i <= 81) OR (i >= 85 AND i <= 87) OR (i >= 91 AND i <= 93) OR (i >= 97 AND i <= 99) THEN
                Return "C";

            !Area B (Robô de Costas para Esteira, à sua Frente
            ELSEIF (i >= 1 AND i <= 9) THEN
                RETURN "B";

            !Area A (Robô de Costas para Esteira, à sua Esquerda
            ELSE
                RETURN "A";
            ENDIF
     ENDFUNC

    !*************************************************************************************************************************
    !Retorna a Posição Específica no Buffer (i= Index Buffer, f= Familia)
    !*************************************************************************************************************************
     FUNC robtarget GetPosicaoBuffer(Num i, Num f)
         VAR robtarget RT_PosicaoBuffer;

         GetDataVal "pBuffer_Pos_" + NumToStr(i, 0) + "_Fam_" + NumToStr(f, 0), RT_PosicaoBuffer;

         RETURN RT_PosicaoBuffer;
     ENDFUNC

    !*************************************************************************************************************************
    !Rotinas de Garra: Abrir (Recuar Servos Para Fora)
    !*************************************************************************************************************************
    PROC GARRA_AbrirGarra()
		!Inicio de ciclo de abertura de garra

        verifica_novamente:
            nNum_Fam := GInput(PN_IN_Numero_Familia);
            WaitTime 0.2;
            SetGO PN_GO_Modelo_Produto, nNum_Fam;
            WaitTime 0.2;

            IF GOutput (PN_GO_Modelo_Produto) = nNum_Fam THEN
                GOTO continue;
            ELSE
                TPWrite "CLP não carregou valor correto para abertura de garra";
                StopMove;
                GOTO verifica_novamente;
            ENDIF

        continue:
            !Revisa se cilindros estão recuados
            WaitDI DI_Fixa_Peça_1_Av, 0\MaxTime:= 5\TimeFlag:=timeout_rc1;
            WaitDI DI_Fixa_Peça_2_Av, 0\MaxTime:= 5\TimeFlag:=timeout_rc2;
            WaitDI DI_Fixa_Peça_1_Rc, 1\MaxTime:= 5\TimeFlag:=timeout_rc3;
            WaitDI DI_Fixa_Peça_2_Rc, 1\MaxTime:= 5\TimeFlag:=timeout_rc4;

            !Se inconsistente, avisa erro:
            IF (timeout_rc1 OR timeout_rc2 OR timeout_rc3 OR timeout_rc4) = TRUE THEN
                PulseDO\PLength:=1, PN_OUT_DO_Cil_NRc;
                TPWrite "Inconsistencia Processo, Travas nao estao recuadas!";
                Stop;
                GOTO continue;
            ENDIF

        !Solicita Abertura de Garra
        SetDO \Sync, PN_OUT_Solicita_Abertura, 1;
        WaitTime 0.5;
        WaitDI PN_IN_Garra_Fechada, 0\MaxTime:= 5\TimeFlag:=timeout_rc1;
        WaitDI PN_IN_Garra_Aberta, 1\MaxTime:= 5\TimeFlag:=timeout_rc2;

        !Se não abriu, avisa erro:
        IF (timeout_rc1 OR timeout_rc2) = TRUE THEN
            PulseDO\PLength:=1, PN_OUT_DO_Cil_NRc;
            SetDO \Sync, PN_OUT_Solicita_Abertura, 0;
            TPWrite "Supervisao Posicionamento Garra, Servos nao Abriram!";
            Stop;
            GOTO continue;
        ENDIF

        SetDO \Sync, PN_OUT_Solicita_Abertura, 0;

	ENDPROC

    !*************************************************************************************************************************
    !Rotinas de Garra: Fechar (Avançar Servos Para o Centro)
    !*************************************************************************************************************************
    PROC GARRA_FecharGarra()
    	!Inicio de ciclo de fechamento de garra

        verifica_novamente:
            nNum_Fam := GInput(PN_IN_Numero_Familia);
            WaitTime 0.2;
            SetGO PN_GO_Modelo_Produto, nNum_Fam;
            WaitTime 0.2;

            IF GOutput (PN_GO_Modelo_Produto) = nNum_Fam THEN
                GOTO continue;
            ELSE
                TPWrite "CLP não carregou valor correto para fechamento de garra";
                StopMove;
                GOTO verifica_novamente;
            ENDIF

        continue:

            !Revisa se cilindros estão recuados
            WaitDI DI_Fixa_Peça_1_Av, 0\MaxTime:= 5\TimeFlag:=timeout_rc1;
            WaitDI DI_Fixa_Peça_2_Av, 0\MaxTime:= 5\TimeFlag:=timeout_rc2;
            WaitDI DI_Fixa_Peça_1_Rc, 1\MaxTime:= 5\TimeFlag:=timeout_rc3;
            WaitDI DI_Fixa_Peça_2_Rc, 1\MaxTime:= 5\TimeFlag:=timeout_rc4;

            !Se inconsistente, avisa erro:
            IF (timeout_rc1 OR timeout_rc2 OR timeout_rc3 OR timeout_rc4) = TRUE THEN
                PulseDO\PLength:=1, PN_OUT_DO_Cil_NRc;
                TPWrite "Inconsistencia Processo, Travas nao estao recuadas!";
                Stop;
                GOTO continue;
            ENDIF

            !Solicita Fechamento Servos:
            SetDO \Sync, PN_OUT_Solicita_Fecha_Garra, 1;
            SetDO\Sync, PN_OUT_Solicita_Abertura, 0;

            WaitDI PN_IN_Garra_Aberta, 0\MaxTime:= 5\TimeFlag:=timeout_av1;
            WaitDI PN_IN_Garra_Fechada, 1\MaxTime:= 5\TimeFlag:=timeout_av2;

            !Se não abriu, avisa erro:
            IF (timeout_av1 OR timeout_av2) = TRUE THEN
                PulseDO\PLength:=1, PN_OUT_DO_Cil_NAv;
                SetDO \Sync, PN_OUT_Solicita_Fecha_Garra, 0;
                TPWrite "Supervisao Posicionamento Garra, Servos nao Fecharam!";
                Stop;
                GOTO continue;
            ENDIF

            SetDO \Sync, PN_OUT_Solicita_Fecha_Garra, 0;
	ENDPROC

    !*************************************************************************************************************************
    !Rotinas de Garra: Travar (Avançar Index Cilindros)
    !*************************************************************************************************************************
    PROC GARRA_TravarProduto()
     init_tp:
        SetDO PN_OUT_DO_Cil_NAv, 0;

        !Trava Produto
        SetDO \Sync, DO_Rc_Fixação_Peça, 0;
        SetDO \Sync, DO_Av_Fixação_Peça, 1;
        !Wait sensores avançado
        WaitTime 1;
        WaitDI DI_Fixa_Peça_1_Rc, 0\MaxTime:= 5\TimeFlag:=timeout_av1;
        WaitDI DI_Fixa_Peça_2_Rc, 0\MaxTime:= 5\TimeFlag:=timeout_av2;
        WaitDI DI_Fixa_Peça_1_Av, 1\MaxTime:= 5\TimeFlag:=timeout_av3;
        WaitDI DI_Fixa_Peça_2_Av, 1\MaxTime:= 5\TimeFlag:=timeout_av4;
        IF (timeout_av1 OR timeout_av2 OR timeout_av3 OR timeout_av4) = TRUE THEN
            PulseDO\PLength:=1, PN_OUT_DO_Cil_NAv;
            TPWrite "Supervisao Sensores, Travas não Avançaram";
            Stop;
            GOTO init_tp;
        ENDIF

    ENDPROC

    !*************************************************************************************************************************
    !Rotinas de Garra: Destravar (Recuar Index Cilindros)
    !*************************************************************************************************************************
    PROC GARRA_DestravarProduto()
    init_dp:
        SetDO PN_OUT_DO_Cil_NRc, 0;

        !Destrava produto na garra
        SetDO \Sync, DO_Av_Fixação_Peça, 0;
        SetDO \Sync, DO_Rc_Fixação_Peça, 1;
        WaitDI DI_Fixa_Peça_1_Av, 0\MaxTime:= 5\TimeFlag:=timeout_rc1;
        WaitDI DI_Fixa_Peça_2_Av, 0\MaxTime:= 5\TimeFlag:=timeout_rc2;
        WaitDI DI_Fixa_Peça_1_Rc, 1\MaxTime:= 5\TimeFlag:=timeout_rc3;
        WaitDI DI_Fixa_Peça_2_Rc, 1\MaxTime:= 5\TimeFlag:=timeout_rc4;
        IF (timeout_rc1 OR timeout_rc2 OR timeout_rc3 OR timeout_rc4) = TRUE THEN
            PulseDO\PLength:=1, PN_OUT_DO_Cil_NRc;
            TPWrite "Supervisao Sensores, Travas não Recuaram";
            Stop;
            GOTO init_dp;
        ENDIF
    ENDPROC

    !*************************************************************************************************************************
    !Rotinas de Garra: Validar Sensor Laser
    !*************************************************************************************************************************
    PROC GARRA_VerificarLaser()
     inicio:
        IF DInput (DI_Pres_Peça_Berço_1) = 0 AND DInput (DI_Pres_Peça_Berço_2) = 1 GOTO Fim;

        PulseDO\PLength:=1, PN_OUT_Produto_Existente;
        TPErase;
        TPWrite "Sensor de presença de peça no berço acionado. Verifique";
        Stop;
        GOTO inicio;

    Fim:
        SetDO PN_OUT_Produto_Existente, 0;
    ENDPROC

    !*************************************************************************************************************************
    !Rotinas de Garra: Validar sensores garra / Garantir que a garra está vazia
    !*************************************************************************************************************************
    PROC GARRA_VerificarGarraVazia()
    !Verifica se robô tem peça na garra ou não

    Verifica:
        IF DI_Pres_Peça_Garra_2 = 1 AND DI_Pres_Peça_Garra_1 = 0 THEN
            GOTO Fim;
        ELSE
            TPErase;
            TPWrite "Deposite manualmente o produto encontrado na garra e reinicie o ciclo";
            TPWrite "Após depositar o produto, adicionar código do produto na IHM";
            IF GInput (PN_IN_Numero_Programa) = 2 THEN
                TPWrite "Programa 'Pega na Esteira de Entrada' necessita de garra vazia para iniciar";
                PulseDO\PLength:=2, PN_OUT_Pos_Home_Manual;
            ELSEIF GInput (PN_IN_Numero_Programa) = 4 THEN
                TPWrite "Programa 'Pega Peça no Buffer' necessita de garra vazia para iniciar";
                PulseDO\PLength:=2, PN_OUT_Pos_Home_Manual;
            ENDIF
            WaitUntil DI_Pres_Peça_Garra_2 = 1 AND DI_Pres_Peça_Garra_1 = 0;
            GOTO Verifica;
        ENDIF
    Fim:
    ENDPROC

    !*************************************************************************************************************************
    !Função para ser chamada pela manutenção (retorno para home)
    !*************************************************************************************************************************
    PROC EXTRAS_PosicionaHomeManual()
        !Movimente manualmente o robô até uma posição em que esteja livre de colisão e acione os comandos abaixo.

    verif:
        pPosição_Atual := CRobT(\Tool:=tGarra \WObj:=wobj0);

        nAux_Limite_Low := 550;
        IF (pPosição_Atual.trans.z > nAux_Limite_Low) THEN
            GOTO DoHome;
        ELSE
            TPErase;
            TPWrite "Posicione Robô mais Alto";
            Stop\NoRegain;
            GOTO verif;
        ENDIF

    DoHome:
        MoveJ pPosição_Trabalho, sMov_Geral_Sem_Produto, fine, tGarra \WObj:=wobj0;
        SetDO PN_OUT_Pos_Home_Manual, 0;


    ENDPROC

    !*************************************************************************************************************************
    !*************************************************************************************************************************
    !*************************************************************************************************************************
    !FUNÇÕES NÃO MAIS UTILIZADAS
    PROC DEPRECATED_VerificacaoInicial ()
        VAR num Passo_Verif_Inic;
        VAR num RespostaTP;
        CONST pos pOffset_Esteiras_Z := [0,0,300];
        CONST pos pOffset_Esteiras_XZ := [100,0,300];

    inicio:

        !Verifica posição atual do robô
        pPosição_Atual := CRobT(\Tool:=tGarra \WObj:=wobj0);

        IF pPosição_Atual.extax.eax_a > 2700 AND pPosição_Atual.trans.x < -1700 THEN
            Passo_Verif_Inic := 10;
            GOTO Analise;
        ENDIF

        IF pPosição_Atual.trans.x < 650 THEN
            Passo_Verif_Inic := 20;
        ENDIF

        IF pPosição_Atual = pHome_Position OR pPosição_Atual = pPosição_Trabalho THEN
            GOTO Final;
        ENDIF

        Passo_Verif_Inic := 30;

   Analise:

        !****************************************************************!
        !               ANALISA O QUE FAZER EM CADA CASO                 !
        !****************************************************************!
        ! Passo_Verif_Inic = 10 - Acima das Esteiras                     !
        ! Passo_Verif_Inic = 20 - Abaixo região segura acima dos berços  !
        ! Passo_Verif_Inic = 30 - Demais regiões                         !
        !****************************************************************!

        TEST Passo_Verif_Inic

        CASE 10:
            !Verifica presença de peça na garra
            IF (DI_Pres_Peça_Garra_2 = 1 AND DI_Pres_Peça_Garra_1 = 0) OR (DI_Pres_Peça_Garra_1 = 1 OR DI_Pres_Peça_Garra_2 = 0 AND DI_Fixa_Peça_1_Rc = 1 AND DI_Fixa_Peça_2_Rc = 1 AND PN_IN_Garra_Aberta = 1) OR (DI_Pres_Peça_Garra_1 = 1 OR DI_Pres_Peça_Garra_2 = 0 AND DI_Fixa_Peça_1_Av = 1 AND DI_Fixa_Peça_2_Av = 1 AND PN_IN_Garra_Fechada = 1) THEN
                GOTO movimento_esteiras;
            ENDIF

            IF DI_Pres_Peça_Garra_1 = 1 OR DI_Pres_Peça_Garra_2 = 0 AND ((DI_Fixa_Peça_1_Rc = 1 OR DI_Fixa_Peça_2_Rc = 1) AND (PN_IN_Garra_Fechada = 1 OR PN_IN_Garra_Aberta = 0)) THEN
                TPReadFK RespostaTP, "Garanta manualmente garra em condições de movimentação e pressione OK", stEmpty, stEmpty, stEmpty, stEmpty, "OK";
                IF (RespostaTP = 5 OR RespostaTP = 0) GOTO inicio;
            ENDIF

    movimento_esteiras:

            pPosição_Desejada := pPosição_Atual;
            pPosição_Desejada.trans := pPosição_Desejada.trans + pOffset_Esteiras_Z;
            MoveL pPosição_Desejada, v30, z10, tGarra \WObj:=wobj0;

            pPosição_Desejada := pPosição_Atual;
            pPosição_Desejada.trans := pPosição_Desejada.trans + pOffset_Esteiras_XZ;
            MoveL pPosição_Desejada, v30, z10, tGarra \WObj:=wobj0;

            GOTO Final;

        CASE 20:
            !Verifica presença de peça na garra
            IF (DI_Pres_Peça_Garra_2 = 1 AND DI_Pres_Peça_Garra_1 = 0) OR (DI_Pres_Peça_Garra_1 = 1 OR DI_Pres_Peça_Garra_2 = 0 AND DI_Fixa_Peça_1_Rc = 1 AND DI_Fixa_Peça_2_Rc = 1 AND PN_IN_Garra_Aberta = 1) OR (DI_Pres_Peça_Garra_1 = 1 OR DI_Pres_Peça_Garra_2 = 0 AND DI_Fixa_Peça_1_Av = 1 AND DI_Fixa_Peça_2_Av = 1 AND PN_IN_Garra_Fechada = 1) THEN
                GOTO movimento_berços;
            ENDIF

            IF DI_Pres_Peça_Garra_1 = 1 OR DI_Pres_Peça_Garra_2 = 0 AND ((DI_Fixa_Peça_1_Rc = 1 OR DI_Fixa_Peça_2_Rc = 1) AND (PN_IN_Garra_Fechada = 1 OR PN_IN_Garra_Aberta = 0))  THEN !Falta sinal garra aberta
                TPReadFK RespostaTP, "Garanta manualmente garra em condições de movimentação e pressione OK", stEmpty, stEmpty, stEmpty, stEmpty, "OK";
                IF (RespostaTP = 5 OR RespostaTP = 0) GOTO inicio;
            ENDIF

        movimento_berços:

            pPosição_Desejada := pPosição_Atual;
            pPosição_Desejada.trans.z := 660;
            MoveL pPosição_Desejada, v30, z10, tGarra \WObj:=wobj0;

            GOTO Final;

        CASE 30:

            !Verifica presença de peça na garra
            IF (DI_Pres_Peça_Garra_2 = 1 AND DI_Pres_Peça_Garra_1 = 0) OR (DI_Pres_Peça_Garra_1 = 1 OR DI_Pres_Peça_Garra_2 = 0 AND DI_Fixa_Peça_1_Rc = 1 AND DI_Fixa_Peça_2_Rc = 1 AND PN_IN_Garra_Aberta = 1) OR (DI_Pres_Peça_Garra_1 = 1 OR DI_Pres_Peça_Garra_2 = 0 AND DI_Fixa_Peça_1_Av = 1 AND DI_Fixa_Peça_2_Av = 1 AND PN_IN_Garra_Fechada = 1) THEN
                GOTO Final;
            ENDIF

            IF DI_Pres_Peça_Garra_1 = 1 OR DI_Pres_Peça_Garra_2 = 0 AND ((DI_Fixa_Peça_1_Rc = 1 OR DI_Fixa_Peça_2_Rc = 1) AND (PN_IN_Garra_Fechada = 1 OR PN_IN_Garra_Aberta = 0))  THEN !Falta sinal garra aberta
                TPReadFK RespostaTP, "Garanta manualmente garra em condições de movimentação e pressione OK", stEmpty, stEmpty, stEmpty, stEmpty, "OK";
                IF (RespostaTP = 5 OR RespostaTP = 0) GOTO inicio;
            ENDIF

        DEFAULT:

            TPErase;
            TPWrite "Não foi possível localizar o robô. Movimente manualmente para a posição inicial";
            Stop;
            GOTO inicio;

        ENDTEST

   Final:
        Passo_Verif_Inic := 0;

        !Se em posição inicial e não foi solicitada parada, encerra rotina
        IF pPosição_Atual = pPosição_Trabalho GOTO Fim;

        !Vai para posição de trabalho
        MoveJ pPosição_Trabalho, sMov_Geral_Com_Produto, fine, tGarra \WObj:=wobj0;

   Fim:
    ENDPROC


    !*************************************************************************************************************************
    !FUNÇÕES EXTRAS: Movimenta Para o Angulo Zero de cada eixo
    !*************************************************************************************************************************
    PROC EXTRAS_MovimentaEixosZero()
      !Ponto Zero do Robo...
      MoveAbsJ [[0,0,0,0,0,0],[0,9E+09,9E+09,9E+09,9E+09,9E+09]] \NoEOffs, v400, fine, tool0;
      !
	ENDPROC

    !*************************************************************************************************************************
    !FUNÇÕES EXTRAS: Teste do 7o eixo
    !*************************************************************************************************************************
    PROC EXTRAS_Teste7oEixo()
        CONST robtarget pPos1:=[[1782.23,-9.35,841.69],[0.0118043,0.0684442,-0.99757,-0.00543028],[-1,0,-1,0],[2708.4,9E+09,9E+09,9E+09,9E+09,9E+09]];
        CONST robtarget pPos2:=[[1782.23,-9.35,841.69],[0.0118043,0.0684442,-0.99757,-0.00543028],[-1,0,-1,0],[-2708.4,9E+09,9E+09,9E+09,9E+09,9E+09]];

        WHILE TRUE DO
            MoveL pPos1, v5000, z50, tGarra\WObj:=wobj0;
            MoveL pPos2, v5000, z50, tGarra\WObj:=wobj0;
        ENDWHILE

    ENDPROC





    !*************************************************************************************************************************
    !*************************************************************************************************************************
    !*************************************************************************************************************************
    !FUNÇÕES NÃO MAIS UTILIZADAS


	PROC DEPRECATED_TesteEixo1()
		MoveJ [[4357.31,-1398.45,1978.14],[0.687563,0.27921,0.236299,0.627265],[-1,0,1,1],[2346.44,9E+09,9E+09,9E+09,9E+09,9E+09]], v2500, z50, tGarra\WObj:=wBuffer_Esq;
		WaitTime\InPos, 1;
		MoveJ [[3711.49,-1299.99,468.29],[0.0309804,-0.747554,-0.66329,0.0158269],[-1,0,1,0],[2346.44,9E+09,9E+09,9E+09,9E+09,9E+09]], v2500, z50, tGarra\WObj:=wBuffer_Esq;
		WaitTime\InPos, 1;
	ENDPROC

    PROC DEPRECATED_Routine1()
		pMov_Pega_Depos_Buffer := pPega_Esteira_Entrada_Fam_1;
        pMov_Pega_Depos_Buffer.trans := pMov_Pega_Depos_Buffer.trans + pOfst_Aprox_Berço_Est_Saida;
        MoveJ pMov_Pega_Depos_Buffer, v1000, fine, tGarra\WObj:=wBuffer_Esq;
        MoveL pPega_Esteira_Entrada_Fam_1, v200, fine, tGarra\WObj:=wBuffer_Esq;
        MoveL pMov_Pega_Depos_Buffer, v2500, fine, tGarra\WObj:=wBuffer_Esq;
        MoveJ pPosição_Trabalho, v1000, fine, tGarra\WObj:=wobj0;
	ENDPROC

    PROC DEPRECATED_TesteAfericao()
      !Ponto de Referencia p/ troca de lagarto..
      MoveJ pCheck_00,v500,z30,tGarra\WObj:=wobj0;
      MoveJ pCheck_01,v500,z30,tGarra\WObj:=wobj0;
      MoveJ pCheck_02,v500,z30,tGarra\WObj:=wobj0;
      MoveL Offs(pCheck,0,0,400),v500,z30,tGarra\WObj:=wobj0;
      MoveL Offs(pCheck,0,0,100), v200, z30, tGarra\WObj:=wobj0;
      MoveL Offs(pCheck,0,0,40), v40, z5, tGarra\WObj:=wobj0;
      MoveL pCheck, v20, fine, tGarra\WObj:=wobj0;
      WaitUntil\InPos,TRUE;
      WaitTime\InPos, 1.5;
      !Stop;
      MoveL Offs(pCheck,0,0,40),v100,z5,tGarra\WObj:=wobj0;
      MoveL Offs(pCheck,0,0,100),v400,z30,tGarra\WObj:=wobj0;
      MoveL Offs(pCheck,0,0,400),v500,z30,tGarra\WObj:=wobj0;
      MoveJ pCheck_02,v500,z30,tGarra\WObj:=wobj0;
      MoveJ pCheck_01,v500,z30,tGarra\WObj:=wobj0;
      MoveJ pCheck_00,v500,z30,tGarra\WObj:=wobj0;
      !
    ENDPROC

ENDMODULE
